// TIA Portal project "AGV75790" (V15)

(* hardware
DEVICE "ET 200S station_1"  ET 200S station
   slot 0: "Rack_0"  Rail
   slot 2: "PLC_AGV75790"  IM 151-8 PN/DP CPU  6ES7 151-8AB01-0AB0  V3.2
      slot 1: "PROFINET interface_1"  PN-IO
         slot 1: "Port_1"  Port
         slot 2: "Port_2"  Port
         slot 3: "Port_3"  Port
   slot 4: "PM-E 24VDC_1"  PM-E 24VDC  6ES7 138-4CA01-0AA0
   slot 5: "8DI x 24VDC_1"  8DI x 24VDC  6ES7 131-4BF00-0AA0
   slot 6: "2AO x U ST_1"  2AO x U ST  6ES7 135-4FB01-0AB0
   slot 7: "8DO x 24VDC / 0.5A_1"  8DO x 24VDC / 0.5A  6ES7 132-4BF00-0AA0
DEVICE "GSD device_1"  GSD.Device.PN
   slot 0: "Rack"  Rack  V1.0
   slot 0: "PGV_AGV75790"  PGVxxx-F200 Position Encoder Color DAP  PGVxxx-F200x-B17-V1D  V1.1.3
      slot 0: "PGVxxx-F200 Position Encoder Color DAP"  PGVxxx-F200 Position Encoder Color DAP
      slot 1: "Interface"  Interface
         slot 1: "Port 1"  Port 1
         slot 2: "Port 2"  Port 2
      slot 1: "Configuration"  Configuration
         slot 0: "Configuration"  Configuration
   slot 3: "status, y-postion, angle, x-position, z-distance"  status, y-postion, angle, x-position, z-distance
      slot 0: "status, y-postion, angle, x-position, z-distance"  status, y-postion, angle, x-position, z-distance
   slot 6: "Status Warning and Error"  Status Warning and Error
      slot 0: "Status Warning and Error"  Status Warning and Error
   slot 7: "input data"  input data
      slot 0: "input data"  input data
DEVICE "GSD device_2"  GSD.Device.PN
   slot 0: "Rack"  Rack  V1.0
   slot 0: "IOLINK_AGV75790"  BNI PNT-508-105-Z015  BNI005H  V3.2
      slot 0: "BNI PNT-508-105-Z015"  BNI PNT-508-105-Z015
      slot 1: "PN-IO"  PN-IO
         slot 1: "port 1 - M12"  port 1 - M12
         slot 2: "port 2 - M12"  port 2 - M12
      slot 1: "IOLINK_AGV72159_1"  BNI PNT-508-105-Z015
         slot 0: "BNI PNT-508-105-Z015"  BNI PNT-508-105-Z015
   slot 2: "MotorDePasso.08Bytes"  IOL_I/O_08/08 byte
      slot 0: "IOL_I/O_08/08 byte"  IOL_I/O_08/08 byte
   slot 3: "Rfid_Bis103"  IOL_I/O_32/32 byte
      slot 0: "IOL_I/O_32/32 byte"  IOL_I/O_32/32 byte
   slot 4: "Standard I/O_3"  Standard I/O
      slot 0: "Standard I/O"  Standard I/O
   slot 5: "Standard I/O_4"  Standard I/O
      slot 0: "Standard I/O"  Standard I/O
   slot 6: "Standard I/O_5"  Standard I/O
      slot 0: "Standard I/O"  Standard I/O
   slot 7: "Standard I/O_6"  Standard I/O
      slot 0: "Standard I/O"  Standard I/O
   slot 8: "Standard I/O_7"  Standard I/O
      slot 0: "Standard I/O"  Standard I/O
   slot 9: "Standard I/O_8"  Standard I/O
      slot 0: "Standard I/O"  Standard I/O
   slot 10: "Station diagnostic"  Station diagnostic
      slot 0: "Station diagnostic"  Station diagnostic
   slot 11: "Sensor supply short circuit"  Sensor supply short circuit
      slot 0: "Sensor supply short circuit"  Sensor supply short circuit
   slot 12: "Periphery error"  Periphery error
      slot 0: "Periphery error"  Periphery error
   slot 13: "Display Leds"  Display Leds
      slot 0: "Display Leds"  Display Leds
DEVICE "SCALANCE X005_1"  SCALANCE X-Station
   slot 0: "SCALANCE X rack"  Rail
   slot 0: "Switch_Rede"  6GK5 008-0GA00-1AB2  V1.0
DEVICE "HMI_AGV75790"  KTP600 Basic color PN
   slot 0: "HMI_AGV75790"  KTP600 Basic color PN  6AV6 647-0AD11-3AX0  12.0.0.0
   slot 1: "HMI_AGV72159"  KTP600 Basic color PN  6AV6 647-0AD11-3AX0  12.0.0.0
   slot 5: "HMI_AGV75790.IE_CP_1"  PROFINET Interface  12.0.0.0
      slot 1: "PROFINET Interface_1"  PROFINET Interface
         slot 1: "Port_1"  Port
*)

// ===== PLC "PLC_AGV75790"  IM 151-8 PN/DP CPU =====

VAR_GLOBAL   // PLC tag table "IO Link"
   "IOLink_StatusAGV" AT %IW80 : Word;   // Status do IOlink 0 - fora da rede, 1 - Na rede
END_VAR

VAR_GLOBAL   // PLC tag table "Entradas"
   "DI_BotaoStart" AT %I0.0 : Bool;   // Botão Wireless de Start do AGV
   "DI_Emergencia" AT %I0.1 : Bool;   // Botão de Emergencia
   "DI_Resevado" AT %I0.2 : Bool;   // Reservado/Sem utilidade no momento
   "DI_Resevado_1" AT %I0.3 : Bool;   // Reservado/Sem utilidade no momento
   "DI_ScannerWarning" AT %I0.4 : Bool;   // Sinal de atenção do Scanner de area
   "DI_ScannerSafety" AT %I0.5 : Bool;   // Sinal de Segurança do Scanner de area
   "DI_Resevado_2" AT %I0.6 : Bool;   // Reservado/Sem utilidade no momento
   "DI_Resevado_3" AT %I0.7 : Bool;   // Reservado/Sem utilidade no momento
END_VAR

VAR_GLOBAL   // PLC tag table "Saidas"
   "AO_MotorTracao" AT %QW752 : Int;   // Sinal de regulagem da velocidade do motor de tração
   "AO_Reservado" AT %QW754 : Int;   // Reservado/Sem utilidade no momento
   "DO_Reservado" AT %Q0.0 : Bool;   // Reservado/Sem utilidade no momento
   "DO_Reservado_1" AT %Q0.1 : Bool;   // Reservado/Sem utilidade no momento
   "DO_Motor.Frente" AT %Q0.2 : Bool;   // Sinal que controla o sentido de giro para frente do motor de tração
   "DO_Motor.Tras" AT %Q0.3 : Bool;   // Sinal que controla o sentido de giro para trás do motor de tração
   "DO_Scanner.Zone1" AT %Q0.4 : Bool;   // Sinal reservado para que seja possivel realizar o aumento e diminuição da area do Scanner de segurança
   "DO_Giroflex" AT %Q0.5 : Bool;   // Sinal luminoso do giroflex - Indica que o AGV está rodando
   "DO_Scanner.Zone2" AT %Q0.6 : Bool;   // Sinal reservado para que seja possivel realizar o aumento e diminuição da area do Scanner de segurança
   "DO_LuzReset" AT %Q0.7 : Bool;   // Sinal luminoso do de emergencia - Indica que o AGV está com o emergencia acionado
END_VAR

VAR_GLOBAL   // PLC tag table "ClockMemory"
   "ClockByte" AT %MB100 : Byte;   // Byte de Clock
   "Clock_10Hz" AT %M100.0 : Bool;   // 100 Milisegundos
   "Clock_5Hz" AT %M100.1 : Bool;   // 200 Milisegundos
   "Clock_2.5Hz" AT %M100.2 : Bool;   // 400 Milisegundos
   "Clock_2Hz" AT %M100.3 : Bool;   // 500 Milisegundos
   "Clock_1.25Hz" AT %M100.4 : Bool;   // 800 Milisegundos
   "Clock_1Hz" AT %M100.5 : Bool;   // 1 Segundos
   "Clock_0.625Hz" AT %M100.6 : Bool;   // 1,6 segundos
   "Clock_0.5Hz" AT %M100.7 : Bool;   // 2 Segundos
END_VAR

VAR_GLOBAL   // PLC tag table "Pgv_Tags"
   "ERR" AT %I1.0 : Bool;   // Error Message, See Error Codes
   "NP" AT %I1.1 : Bool;   // No Absolute Position
   "WRN" AT %I1.2 : Bool;   // Warning Present, See Warning Module
   "CC" AT %I1.3 : Bool;   // Control Code Detected
   "Reservado" AT %I1.4 : Bool;   // Reserved
   "FR" AT %I1.5 : Bool;   // Follow Right-hand lane
   "FL" AT %I1.6 : Bool;   // Follow Left-hand lane
   "NL" AT %I1.7 : Bool;   // No lane detected
   "RP" AT %I2.0 : Bool;   // Relative Position
   "LC" AT %I2.1 : Bool;   // Bit field LSB, Number of detected lanes
   "LC_1" AT %I2.2 : Bool;   // Bit field MSB, Number of detected lanes
   "TA" AT %I2.3 : Bool;   // Data Matrix tag present
   "Reservado_1" AT %I2.4 : Bool;   // Reserved
   "Reservado_2" AT %I2.5 : Bool;   // Reserved
   "Reservado_3" AT %I2.6 : Bool;   // Reserved
   "Reservado_4" AT %I2.7 : Bool;   // Reserved
   "PositionY" AT %ID3 : DWord;   // Posição no eixo Y
   "Angle" AT %IW8 : Word;   // Angulo
   "PositionX" AT %ID10 : DWord;   // Posição no eixo X
   "PositionZ" AT %IW14 : Word;   // Posição no eixo Z
   "Output_Data" AT %QB1 : Byte;   // Dados de Saida
   "Status" AT %ID15 : DWord;   // Status PGV
   "Erro" AT %IW20 : Word;   // Erros PGV
END_VAR

TYPE "DT_FML_STATUS"
VERSION : 0.1
   STRUCT
      Err : Bool;
      Cat : Int;
      ID : DInt;
   END_STRUCT;
END_TYPE

TYPE "DT_FML_PRM_FILE"
VERSION : 0.1
// DT_FML_PRM_FILE_TRANSFER
   STRUCT
      Control : Int;
      BitSequenceNr : Int;
      Data : Array[1..6] of Byte;
   END_STRUCT;
END_TYPE

TYPE "DT_FML_REF"
// DT_FML_PRM_REF
   STRUCT
      InData : Struct
         FHPP : Array[1..8] of Byte;
         FPC : Array[1..8] of Byte;
         FHPPplus : Array[1..10] of DInt;
      END_STRUCT;
      OutData : Struct
         FHPP : Array[1..8] of Byte;
         FPC : Array[1..8] of Byte;
         FHPPplus : Array[1..10] of DInt;
      END_STRUCT;
      Modbus : Bool;
      DeviceType : String[16];
      DeviceTypeNo : Byte;
      MemberID : Int;   // Current Axis-ID
      MemberIDmax : Int;   // Maximum Axis-ID
      Done : Bool;   // Execution Done
      Err : Bool;   // Fault occured
      PNU : Word;   // Number of the Parameter
      ActPNU : Word;   // Actual Number of the Parameter
      ReqID : Int;   // Read upper Limit of the Parameter
      RespID : Int;   // Read lower limit of the Parameter
      FPCC_Modus : Byte;   // modus of parameter channel control
      FPCS_Modus : Byte;   // modus of parameter channel status
      FPCC_Packet : "DT_FML_PRM_FILE";
      FPCS_Packet : "DT_FML_PRM_FILE";
      Subindex : Byte;   // Subindex of the Parameter to Exchange
      ActSubindex : Byte;   // Actual Subindex of the Parameter
      DatatypeWR : Byte;   // Length of the Parameter to Exchange in Byte
      DatatypeRD : Byte;   // Actual Length of the Parameter in Byte
      ParamValueWR : DInt;   // Value of the Parameter to Exchange
      ParamValueRD : DInt;   // Read Value of Parameter
   END_STRUCT;
END_TYPE

TYPE "EscritaTakt"
   STRUCT
      Emergencia : Bool;   // Botao de Emergecencia
      Warning : Bool;   // Area de Warning do Scanner
      Safety : Bool;   // Area de Safety do Scanner
      ConectarTakt : Bool;   // 0 - Desconectado / 1 - Conectado
      Rodando : Bool;
      Falha : Bool;
      AutomaticoManual : Byte;   // 1 - Manual / 2 - Automatico
      VelocidadeAtual : Int;   // Velocidade Atual
      Posto : Byte;   // Posto em que o AGV está
      Comando : Byte;   // Ultimo comando
      Velocidade : Byte;   // Velocidade Setada
      Processo : Byte;   // 1 - Ecu / 2 - SKD
      "Erros.Agv" : Byte;   // 0 á 256, cada numero um erro. 1 - Tudo Ok
      "Erros.Pgv" : Byte;   // 0 á 256, cada numero um erro. 1 - Tudo Ok
      "Erros.Rfid" : Byte;   // 0 á 256, cada numero um erro. 1 - Tudo Ok
      "Erros.MotorPasso" : Byte;   // 0 á 256, cada numero um erro. 1 - Tudo Ok
      "Erros.IOLink" : Byte;   // 0 á 256, cada numero um erro. 1 - Tudo Ok
      "Erros.Comunicacao" : Byte;   // 0 á 256, cada numero um erro. 1 - Tudo Ok
      Reservado : Byte;   // Reservado
      Reservado_1 : Byte;   // Reservado
      Reservado_2 : Byte;   // Reservado
      Reservado_3 : Byte;   // Reservado
      Reservado_4 : Byte;   // Reservado
      Reservado_5 : Byte;   // Reservado
      Reservado_6 : Byte;   // Reservado
      Reservado_7 : Byte;   // Reservado
      Reservado_8 : Byte;   // Reservado
   END_STRUCT;
END_TYPE

TYPE "LeituraTakt"
   STRUCT
      EmergenciaECU : Bool;   // Emergencia
      EmergenciaSKD : Bool;   // Emergencia
      StartAgvECU : Bool;   // Start by takt
      StopAgvECU : Bool;   // Stop by takt
      StartAgvSKD : Bool;   // Start by takt
      StopAgvSKD : Bool;   // Stop by takt
      WatchDog : Bool;   // WatchDog
      TOD : Time_Of_Day;   // Time of day
   END_STRUCT;
END_TYPE

// folder: 01_Controle/02_DB

DATA_BLOCK "DB1_DatabaseAgv"   // DB1
TITLE = DB1_DatabaseAgv
{ S7_Optimized_Access := 'FALSE' }
AUTHOR : ssbjvq
VERSION : 0.1
// Está DB é responsavel por centralizar toda a informação do AGV
   VAR
      Entradas : Struct   // Sinais do cartão de entrada digital
         BotaoStart : Bool;   // Botão Wireless de Start do AGV
         BotaoEmergencia : Bool;   // Botão de Emergencia
         ScannerWarning : Bool;   // Sinal de atenção do Scanner de area
         ScannerSafety : Bool;   // Sinal de Segurança do Scanner de area
         Reservada_4 : Bool;   // Reservado/Sem utilidade no momento
         Reservada_5 : Bool;   // Reservado/Sem utilidade no momento
         Reservada_6 : Bool;   // Reservado/Sem utilidade no momento
      END_STRUCT;
      Saidas : Struct   // Sinais dos cartões de saida
         MotorFrente : Bool;   // Sinal que controla o sentido de giro para frente do motor de tração
         MotorTras : Bool;   // Sinal que controla o sentido de giro para trás do motor de tração
         Zona1_Scanner : Bool;   // Sinal reservado para que seja possivel realizar o aumento e diminuição da area do Scanner de segurança
         Zona2_Scanner : Bool;   // Sinal luminoso do giroflex - Indica que o AGV está rodando
         Giroflex : Bool;   // Sinal reservado para que seja possivel realizar o aumento e diminuição da area do Scanner de segurança
         LuzReset : Bool;   // Sinal luminoso do de emergencia - Indica que o AGV está com o emergencia acionado
         Reservada : Bool;   // Reservado/Sem utilidade no momento
         VelocidadeMotorTracao : Int;   // Sinal de regulagem da velocidade do motor de tração
         Analog_1 : Int;   // Reservado/Sem utilidade no momento
      END_STRUCT;
      PGV : Struct   // Sinais do PGV
         Module2 : Struct
            Status : Struct
               ERR : Bool;   // Error Message, See Error Codes
               NP : Bool;   // No Absolute Position
               WRN : Bool;   // Warning Present, See Warning Module
               CC : Bool;   // Control Code Detected
               Reservado : Bool;   // Reserved
               FR : Bool;   // Follow Right-hand lane
               FL : Bool;   // Follow Left-hand lane
               NL : Bool;   // No lane detected
               RP : Bool;   // Relative Position
               LC : Bool;   // Bit field LSB, Number of detected lanes
               LC_1 : Bool;   // Bit field MSB, Number of detected lanes
               TA : Bool;   // Data Matrix tag present
               Reservado_1 : Bool;   // Reserved
               Reservado_2 : Bool;   // Reserved
               Reservado_3 : Bool;   // Reserved
               Reservado_4 : Bool;   // Reserved
            END_STRUCT;
            PositionY : DWord;
            Angle : Word;
            PositionX : DWord;
            PositionZ : Word;
         END_STRUCT;
         Module5 : Struct
            Status : Word;
            BitmaskWarning : Word;
            ErroNumber : Word;
         END_STRUCT;
         Mensagens : String;
         NaRota : Bool;
         Rota : Byte := 16#0A;
      END_STRUCT;
      RFID : Struct   // Sinais do RFID
         Inputs : Struct
            Init : Bool;   // Deve ser pulsado para iniciar a leitura
            Start : Bool;   // Deve ser dado o start para o RIFD funcionar
            Reset : Bool;   // Reseta se existe problema
            HeadOff : Bool;
            Dynamic : Bool;
            HW_IO : Int := 80;   // Endereço do dispositivo na rede
            Command : Int := 1;   // Comando 1 - Leitura / 2 - Escrita
            DB_Send : Int := 421;   // Numero da DB de envio de dados
            Offset_DBSend : Int := 0;   // Deslocamento de bits da DB de envio
            DB_Receive : Int := 420;   // Numero da DB de recebimento de dados
            Offset_DBReceive : Int := 0;   // Deslocamento de bits da DB de recebimento
            StartAddress : Int := 0;   // Primeiro endereço a ser lido
            NumberOfByte : Int := 32;   // Numero de bytes a ser lidos até 32 bits
            Watchdog : S5Time := S5T#100ms;
         END_STRUCT;
         Posto : Int;   // Valor do posto
         Comando : Int;   // Valor do comando
         Velocidade : Int := 22;   // Valor da velocidade
         Processo : Int;   // Valor da linha
         Error : Bool;   // Sinal de erro
         TagPresente : Bool;   // Sinal de Tag presente
         CodigoErro : Int;   // Codigo do erro
         Ready : Bool;   // Sinal de Pronto para uso
         Fault : Bool;   // Sinal de falha
         Mensagens : String;   // Mensagens de falha
      END_STRUCT;
      MotorDePasso : Struct   // Sinais do Motor de Passo
         GetIO : Struct   // Bloco de comunicação
            Inputs : Struct
               IAddress_FHPP : Word := 16#46;   // Endereço do dispositivo em HEX
               Offset : Int := 0;   // Deslocamento de bits
               DeviceType : String[16] := 'CMMO_ST';   // Tipo do dispositivo
            END_STRUCT;
            Outputs : Struct
               Error : Bool;   // Sinal de falha na comunicação
               Status : "DT_FML_STATUS";   // Status de leitura
            END_STRUCT;
         END_STRUCT;
         SetIO : Struct   // Bloco de comunicação
            Inputs : Struct
               ID : Word := 16#46;   // Endereço do dispositivo em HEX
               Offset : Int;   // Deslocamento de bits
            END_STRUCT;
            Outputs : Struct
               Error : Bool;   // Sinal de falha na comunicação
               Status : "DT_FML_STATUS";   // Status de leitura
            END_STRUCT;
         END_STRUCT;
         Inputs : Struct   // Sinais de entrada
            EnableDrive : Bool;   // Habilitar drive
            Stop : Bool;   // Parar motor
            Halt : Bool;
            Brake : Bool;   // Freio do motor
            ResetFault : Bool;   // Resetar falha do motor
            HMIAccessLocked : Bool;   // Travar acesso via IHM
            OPM : Int;   // Modo de operação
            StartTask : Bool;   // Iniciar tarefa
            StartHoming : Bool;   // Iniciar homing
            JogPos : Bool;   // Virar a esquerda
            JogNeg : Bool;   // Virar a direita
            TeachActValue : Bool;
            ClearRemPos : Bool;
            Relative : Bool;
            DeactivateStrokeLimit : Bool;   // Desativar limite de giro
            ExecuteFunction : Bool;   // Executar função gravada
            RecordNo : Int;   // Numero da função
            SetFunctionNumber : Int;   // Setar numero da função
            SetFunctionGroup : Int;   // Setar numero do grupo de funções
            SetValueVelocity : DInt;   // Setar valor de velocidade do motor
            SetValuePosition : DInt;   // Setar valor de posição
            SetValueForceRamp : DInt;   // Setar valor de rampa de força
            SetValueForce : DInt;   // Setar valor de força
            SetValueRotRamp : DInt;   // Setar valor de rampa de rotação
            SetValueRotSpeed : DInt;   // Setar valor de rotação
         END_STRUCT;
         OutPuts : Struct   // Sinais de saidas
            DriveEnabled : Bool;   // Drive habilitado
            Ready : Bool;   // Pronto para rodar
            Warning : Bool;   // Em modo atenção
            Fault : Bool;   // Em falha
            SupplyVoltPresent : Bool;   // Tensão presente
            ControlFCT_HMI : Bool;   // Controle via IHM
            StateOPM : Int;   // Status do modo de operação
            HaltNotActive : Bool;   // Halt não ativado
            AckStart : Bool;   // Movimento iniciado
            MC : Bool;   // Movimento Completo
            AckTeach : Bool;
            DriveMoving : Bool;   // Motor em movimento
            DragError : Bool;   // Error de movimentação
            StandStillControl : Bool;
            HomingValid : Bool;   // Homing valido
            ActualRecordNo : Int;   // Numero de gravação atual
            RC1 : Bool;
            RCC : Bool;
            VelocityLimitReached : Bool;   // Velocidade limite atingida
            StrokeLimitReached : Bool;   // Giro limite atingido
            FunctionIsActive : Bool;   // Modo função ativado
            ActualFunctionNumber : Int;   // Numero atual da função
            ActualFunctionGroup : Int;   // Numero atual do grupo de função
            ActualPosition : DInt;   // Posição atual
            ActualVelocity : Int;   // Velocidade atual
            ActualForce : Int;   // Força atual
            ActualRotRamp : Int;   // Rampa de rotação atual
            ActualRotSpeed : DInt;   // Velocidade de rotação atual
         END_STRUCT;
         Mensagens : String;   // Mensagens de motor de passo
      END_STRUCT;
      IOLink : Struct   // Sinais do IOLink
         Mensagens : String;   // Mensagens de falha do IO Link
      END_STRUCT;
      Takt : Struct   // Sinais do Takt
         Mensagens : String;
      END_STRUCT;
      Mensagens : String;   // Mensagens gerais do AGV
   END_VAR
BEGIN
END_DATA_BLOCK

DATA_BLOCK "DB3_Memorias"   // DB3
{ S7_Optimized_Access := 'FALSE' }
VERSION : 0.1
   VAR
      StartStop : Bool;   // Memoria de Start ou Stop
      Rfid : Struct   // Memorias do RFId
         PararAgv : Bool;   // Memoria de parada do AGV
         Comando : Int;   // Memoria de comando
         Velocidade : Int;   // Memoria de velocidade
         Linha : Int;   // Memoria de linha
         Posto : Int;   // Memoria de posto
         LeituraEscrita : Int;   // Memoria de leitura 1 ou escrita 2
      END_STRUCT;
      Pgv : Struct   // Memorias do Pgv
         NaRota : Bool;   // AGV na rota
         Angulo : Int;   // Angulo
         Direita : Bool;   // Direita
         Esquerda : Bool;   // Esquerda
      END_STRUCT;
      Frente : Bool;
      Tras : Bool;
      Esquerda : Bool;
      Direita : Bool;
      Posicao : DInt;   // Posição motor de passo
      Velocidade : Int;   // Velocidade
      EmCurva : Bool;   // Memoria Em curva
      EmCurvaIntermediario : Bool;   // Memoria Em curva intermediario
      LimiteGiroDireita : Bool;   // Bloco de comunicação
      LimiteGiroEsquerda : Bool;   // Memoria de limite de giro
   END_VAR
BEGIN
END_DATA_BLOCK

DATA_BLOCK "DB100_ManualAutomatico_DB"   // DB100
{ S7_Optimized_Access := 'FALSE' }
VERSION : 0.1
// stored: InstanceOfName FB100_ManualAutomatico
"FB100_ManualAutomatico"
BEGIN
END_DATA_BLOCK

DATA_BLOCK "DB102_AgvStartStop"   // DB102
{ S7_Optimized_Access := 'FALSE' }
VERSION : 0.1
// stored: InstanceOfName FB102_AgvStartStop
"FB102_AgvStartStop"
BEGIN
END_DATA_BLOCK

DATA_BLOCK "DB105_Sinalizacao"   // DB105
{ S7_Optimized_Access := 'FALSE' }
VERSION : 0.1
// stored: InstanceOfName FB105_Sinalizacao
"FB105_Sinalizacao"
BEGIN
END_DATA_BLOCK

// folder: 02_MotorPasso/02_DB

DATA_BLOCK "DB200_ControleMotorDePasso"   // DB200
{ S7_Optimized_Access := 'FALSE' }
VERSION : 0.1
// stored: InstanceOfName FB200_ControleMotorDePasso
"FB200_ControleMotorDePasso"
BEGIN
END_DATA_BLOCK

// folder: 03_Pgv/02_DB

DATA_BLOCK "DB301_PgvDados"   // DB4
{ S7_Optimized_Access := 'FALSE' }
VERSION : 0.1
// stored: InstanceOfName FB301_PgvDados
"FB301_PgvDados"
BEGIN
END_DATA_BLOCK

DATA_BLOCK "DB300_LogicaPgv"   // DB300
{ S7_Optimized_Access := 'FALSE' }
VERSION : 0.1
// stored: InstanceOfName FB300_LogicaPgv
"FB300_LogicaPgv"
BEGIN
END_DATA_BLOCK

// folder: 04_Rfid/02_DB

DATA_BLOCK "DB400_LogicaRfid"   // DB400
{ S7_Optimized_Access := 'FALSE' }
VERSION : 0.1
// stored: InstanceOfName FB400_LogicaRfid
"FB400_LogicaRfid"
BEGIN
END_DATA_BLOCK

DATA_BLOCK "DB420_LeituraRfid"   // DB420
{ S7_Optimized_Access := 'FALSE' }
VERSION : 0.1
   VAR
      RfidLeitura : Array[0..31] of Int;
   END_VAR
BEGIN
   RfidLeitura[3] := 22;   // Velocidade
   RfidLeitura[1] := 2;   // Posto de trabalho
   // RfidLeitura[2] : Comando
   // RfidLeitura[4] : Linha/Processo
   // RfidLeitura[0] : Não utilizado
   // RfidLeitura[5] : Não utilizado
   // RfidLeitura[6] : Não utilizado
   // RfidLeitura[7] : Não utilizado
   // RfidLeitura[8] : Não utilizado
   // RfidLeitura[9] : Não utilizado
   // RfidLeitura[10] : Não utilizado
   // RfidLeitura[11] : Não utilizado
   // RfidLeitura[12] : Não utilizado
   // RfidLeitura[13] : Não utilizado
   // RfidLeitura[14] : Não utilizado
   // RfidLeitura[15] : Não utilizado
   // RfidLeitura[16] : Não utilizado
   // RfidLeitura[17] : Não utilizado
   // RfidLeitura[18] : Não utilizado
   // RfidLeitura[19] : Não utilizado
   // RfidLeitura[20] : Não utilizado
   // RfidLeitura[21] : Não utilizado
   // RfidLeitura[22] : Não utilizado
   // RfidLeitura[23] : Não utilizado
   // RfidLeitura[24] : Não utilizado
   // RfidLeitura[25] : Não utilizado
   // RfidLeitura[26] : Não utilizado
   // RfidLeitura[27] : Não utilizado
   // RfidLeitura[28] : Não utilizado
   // RfidLeitura[29] : Não utilizado
   // RfidLeitura[30] : Não utilizado
   // RfidLeitura[31] : Não utilizado
END_DATA_BLOCK

DATA_BLOCK "DB421_EscritaRfid"   // DB421
{ S7_Optimized_Access := 'FALSE' }
VERSION : 0.1
   VAR
      RfidEscrita : Array[0..31] of Int;
   END_VAR
BEGIN
   // RfidEscrita[0] : Não utilizado
   // RfidEscrita[1] : Posto de trabalho
   // RfidEscrita[2] : Comando
   // RfidEscrita[3] : Velocidade
   // RfidEscrita[4] : Linha/Processo
   // RfidEscrita[5] : Não utilizado
   // RfidEscrita[6] : Não utilizado
   // RfidEscrita[7] : Não utilizado
   // RfidEscrita[8] : Não utilizado
   // RfidEscrita[9] : Não utilizado
   // RfidEscrita[10] : Não utilizado
   // RfidEscrita[11] : Não utilizado
   // RfidEscrita[12] : Não utilizado
   // RfidEscrita[13] : Não utilizado
   // RfidEscrita[14] : Não utilizado
   // RfidEscrita[15] : Não utilizado
   // RfidEscrita[16] : Não utilizado
   // RfidEscrita[17] : Não utilizado
   // RfidEscrita[18] : Não utilizado
   // RfidEscrita[19] : Não utilizado
   // RfidEscrita[20] : Não utilizado
   // RfidEscrita[21] : Não utilizado
   // RfidEscrita[22] : Não utilizado
   // RfidEscrita[23] : Não utilizado
   // RfidEscrita[24] : Não utilizado
   // RfidEscrita[25] : Não utilizado
   // RfidEscrita[26] : Não utilizado
   // RfidEscrita[27] : Não utilizado
   // RfidEscrita[28] : Não utilizado
   // RfidEscrita[29] : Não utilizado
   // RfidEscrita[30] : Não utilizado
   // RfidEscrita[31] : Não utilizado
END_DATA_BLOCK

// folder: 05_Ihm/02_DB

DATA_BLOCK "DB500_SinaisIhm"   // DB500
{ S7_Optimized_Access := 'FALSE' }
VERSION : 0.1
   VAR
      ManualAutomatico : Int := 1;   // 1 Modo manual/ 2 - modo automatico
      Start : Bool;   // Botão de Start IHM
      Processo : Int := 1;   // Botão de processo IHM
      VelocidadeManual : Int := 18;   // Velocidade em manual
      VelocidadeWarning : Int := 10;   // Velocidade em Warning
      ResetFault : Bool;   // Botao de Resetar falha do motor
      ManFrente : Bool;   // Botao manual frente
      ManTras : Bool;   // Botao manual tras
      ManDireita : Bool;   // Botao manual direita
      ManEsquerda : Bool;   // Botao manual esquerda
      ConexaoTakt : Bool := TRUE;   // Conectar com o takt
      PostoRfid : Int;   // Input de gravação de tag
      ComandoRfid : Int;   // Input de gravação de tag
      VelocidadeRfid : Int;   // Input de gravação de tag
      ProcessoRfid : Int;   // Input de gravação de tag
      LeituraEscritaRfid : Bool;   // Modo de operação do RFID
      VelocidadeAutomatico : Int := 15;   // Valor de velocidade em automatico
      VelocidadeAtual : Int;   // Valor de velocidade atual
      ConectarTakt : Int := 1;   // 1 - Conecta com o Takt / 0 - Desconectado
      ResetFalha_Rfid : Bool := False;   // Resetar falha RFID
   END_VAR
BEGIN
END_DATA_BLOCK

// folder: 06_Errors/02_DB

DATA_BLOCK "DB600_AgvSinais"   // DB600
{ S7_Optimized_Access := 'FALSE' }
VERSION : 0.1
   VAR
      Inputs : Struct   // Cartão de entrada
         "8DI_24V" : Struct   // Cartão de entrada
            "I0.0" : Bool;   // Botão Wireless de Start do AGV
            "I0.1" : Bool;   // Botão de Emergencia
            "I0.2" : Bool;   // Reservado/Sem utilidade no momento
            "I0.3" : Bool;   // Reservado/Sem utilidade no momento
            "I0.4" : Bool;   // Sinal de atenção do Scanner de area
            "I0.5" : Bool;   // Sinal de Segurança do Scanner de area
            "I0.6" : Bool;   // Reservado/Sem utilidade no momento
            "I0.7" : Bool;   // Reservado/Sem utilidade no momento
         END_STRUCT;
      END_STRUCT;
      Outputs : Struct   // Cartões de saida
         "8DO_24V" : Struct   // Cartão Digital
            "Q0.0" : Bool;   // Reservado/Sem utilidade no momento
            "Q0.1" : Bool;   // Reservado/Sem utilidade no momento
            "Q0.2" : Bool;   // Sinal que controla o sentido de giro para frente do motor de tração
            "Q0.3" : Bool;   // Sinal que controla o sentido de giro para trás do motor de tração
            "Q0.4" : Bool;   // Sinal reservado para que seja possivel realizar o aumento e diminuição da area do Scanner de segurança
            "Q0.5" : Bool;   // Sinal luminoso do giroflex - Indica que o AGV está rodando
            "Q0.6" : Bool;   // Sinal reservado para que seja possivel realizar o aumento e diminuição da area do Scanner de segurança
            "Q0.7" : Bool;   // Sinal luminoso do de emergencia - Indica que o AGV está com o emergencia acionado
         END_STRUCT;
         "2AO x U ST" : Struct   // Cartão Analogico
            QW750 : Word;   // Sinal de regulagem da velocidade do motor de tração
            QW752 : Word;   // Reservado/Sem utilidade no momento
         END_STRUCT;
      END_STRUCT;
      RFID : Struct   // Sinais RFID
         Posto : Int;   // Valor do posto
         Comando : Int;   // Valor do comando
         Velocidade : Int;   // Valor da velocidade
         Linha : Int;   // Valor da linha
         Tag_Presente : Bool;   // Sinal de erro
         Error : Bool;   // Sinal de Tag presente
         Code_Error : Int;   // Codigo do erro
         Ready : Bool;   // Sinal de Pronto para uso
         Mensagem : String;   // Sinal de falha
      END_STRUCT;
      Stepping_Motor : Struct   // Sinais Motor de Passo
         Inputs : Struct   // Entrada
            Enabla_Drive : Bool;   // Habilitar Dirve
            Stop : Bool;   // Parado
            "Start Task" : Bool;   // Inicia Tarefa
            Opm : Int;   // Modo de operação
            Brake : Bool;   // Freio
         END_STRUCT;
         Outputs : Struct   // Saidas
            DriveEnabled : Bool;   // Drive habilitado
            Ready : Bool;   // Pronto para rodar
            Warning : Bool;   // Em modo atenção
            Fault : Bool;   // Em falha
            SupplyVoltPresent : Bool;   // Tensão presente
            DragError : Bool;   // Error de movimentação
            HomingValid : Bool;   // Homing valido
            StrokeLimitReached : Bool;   // Giro limite atingido
            ActualPosition : DInt;   // Posição atual
         END_STRUCT;
         Mensagem : String;   // Mensagens do motor de passo
      END_STRUCT;
      PGV : Struct   // Sinais PGV
         Mensagem : String;   // Mensagens do PGV
         ERR : Bool;   // Error Message, See Error Codes
         NP : Bool;   // No Absolute Position
         WRN : Bool;   // Warning Present, See Warning Module
         CA : Bool;   // Control Code Detected
         FR : Bool;   // Reserved
         FL : Bool;   // Follow Right-hand lane
         NL : Bool;   // Follow Left-hand lane
         RP : Bool;   // No lane detected
         TA : Bool;   // Relative Position
         PositionData_Y : Int;   // Bit field LSB, Number of detected lanes
         PositionData_X : Int;   // Bit field MSB, Number of detected lanes
         PositionData_Z : Int;   // Data Matrix tag present
         AngleData : Int;   // Angulo
         "DataMatrix.CCStatus" : Byte;
         "DataMatrix.CCNumber" : Word;
         "DataMatrix.TagNumber" : DWord;
         BitmaskWarning : Word;
         ErrorNumber : Word;
         "OUT_Warning.Monitoring" : Word;
         "OUT_Error.Monitoring" : Word;
      END_STRUCT;
      DateHora : Date_And_Time;   // Data e Hora
      Mensagens_Global : String;   // Mensagens de falha
      Alarms : Array[0..8] of Int;   // Alarmes na lista
   END_VAR
BEGIN
   // Alarms[0] : PGV
   // Alarms[1] : RFID
   // Alarms[2] : MOTOR DE PASSO
   // Alarms[3] : PLC
   // Alarms[4] : IO-LINK
   // Alarms[5] : SINAIS - 0 - Emergencia, 1 - Warning, 2- Safety, 3 - Fora da rota,
END_DATA_BLOCK

DATA_BLOCK "DB603_StatusGeralAgv"   // DB603
{ S7_Optimized_Access := 'FALSE' }
VERSION : 0.1
// stored: InstanceOfName FB603_StatusGeralAgv
"FB603_StatusGeralAgv"
BEGIN
END_DATA_BLOCK

// folder: 07_Takt/02_DB

DATA_BLOCK "DB700_EnviaDados"   // DB700
TITLE = DB700_EnviaDados
{ S7_Optimized_Access := 'FALSE' }
AUTHOR : ssbjvq
VERSION : 0.1
// DB700_EnviaDados
   VAR
      Dados : "EscritaTakt";
   END_VAR
BEGIN
END_DATA_BLOCK

DATA_BLOCK "DB701_RecebeDados"   // DB701
TITLE = DB701_RecebeDados
{ S7_Optimized_Access := 'FALSE' }
AUTHOR : ssbjvq
VERSION : 0.1
// DB701_RecebeDados
   VAR
      Dados : "LeituraTakt";
   END_VAR
BEGIN
END_DATA_BLOCK

DATA_BLOCK "DB703_ControleTakt"   // DB703
{ S7_Optimized_Access := 'FALSE' }
AUTHOR : ssbjvq
VERSION : 0.1
// stored: InstanceOfName FB703_ControleTakt
"FB703_ControleTakt"
BEGIN
END_DATA_BLOCK

DATA_BLOCK "DB704_DadosTakt"   // DB704
{ S7_Optimized_Access := 'FALSE' }
VERSION : 0.1
   VAR
      Dados_Takt : Struct
         Tempo_Takt : DInt;
         Tempo_StopTime : DInt;
         Objetivo : Int;
         Atual : Int;
         Andons : Array[0..8] of Bool;
      END_STRUCT;
   END_VAR
BEGIN
END_DATA_BLOCK

// folder: (top level)

ORGANIZATION_BLOCK "Main"   // OB1, LAD
TITLE = "Main Program Sweep (Cycle)"
{ S7_Optimized_Access := 'FALSE' }
VERSION : 0.1
// Bloco principal do CLP, ele é responsavel por rodar toda a logica do CLP e organizar o programa.
   VAR_TEMP
      OB1_EV_CLASS : Byte;   // Bits 0-3 = 1 (Coming event), Bits 4-7 = 1 (Event class 1)
      OB1_SCAN_1 : Byte;   // 1 (Cold restart scan 1 of OB 1), 3 (Scan 2-n of OB 1)
      OB1_PRIORITY : Byte;   // Priority of OB Execution
      OB1_OB_NUMBR : Byte;   // 1 (Organization block 1, OB1)
      OB1_RESERVED_1 : Byte;   // Reserved for system
      OB1_RESERVED_2 : Byte;   // Reserved for system
      OB1_PREV_CYCLE : Int;   // Cycle time of previous OB1 scan (milliseconds)
      OB1_MIN_CYCLE : Int;   // Minimum cycle time of OB1 (milliseconds)
      OB1_MAX_CYCLE : Int;   // Maximum cycle time of OB1 (milliseconds)
      OB1_DATE_TIME : Date_And_Time;   // Date and time OB1 started
   END_VAR
BEGIN

REGION Network 1: Modo Automatico ou Manual
   // Este bloco é responsavel por realizar o controle do AGV no modo automatico e no modo manual, sem ele o AGV não realiza nenhum movimento.
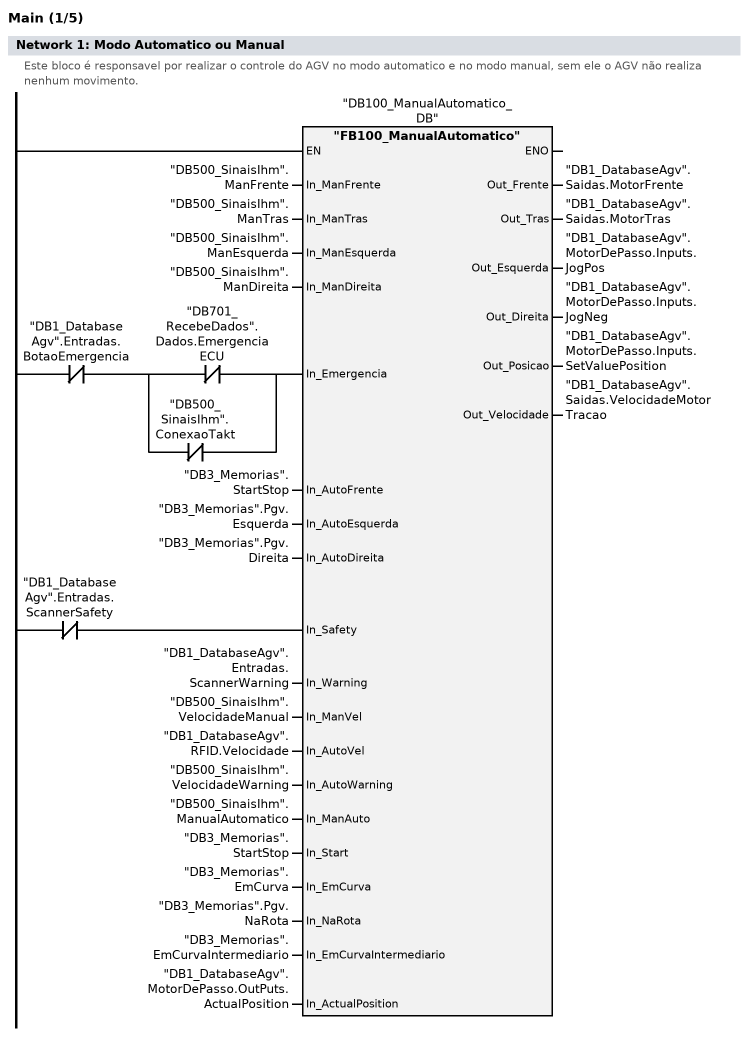
   RUNG wire#powerrail
      "DB100_ManualAutomatico_DB"(In_Emergencia := wire#w2, In_Safety := wire#w3, In_ManFrente := "DB500_SinaisIhm".ManFrente, In_ManTras := "DB500_SinaisIhm".ManTras, In_ManEsquerda := "DB500_SinaisIhm".ManEsquerda, In_ManDireita := "DB500_SinaisIhm".ManDireita, In_AutoFrente := "DB3_Memorias".StartStop, In_AutoEsquerda := "DB3_Memorias".Pgv.Esquerda, In_AutoDireita := "DB3_Memorias".Pgv.Direita, In_Warning := "DB1_DatabaseAgv".Entradas.ScannerWarning, In_ManVel := "DB500_SinaisIhm".VelocidadeManual, In_AutoVel := "DB1_DatabaseAgv".RFID.Velocidade, In_AutoWarning := "DB500_SinaisIhm".VelocidadeWarning, In_ManAuto := "DB500_SinaisIhm".ManualAutomatico, In_Start := "DB3_Memorias".StartStop, In_EmCurva := "DB3_Memorias".EmCurva, In_NaRota := "DB3_Memorias".Pgv.NaRota, In_EmCurvaIntermediario := "DB3_Memorias".EmCurvaIntermediario, In_ActualPosition := "DB1_DatabaseAgv".MotorDePasso.OutPuts.ActualPosition, Out_Frente => "DB1_DatabaseAgv".Saidas.MotorFrente, Out_Tras => "DB1_DatabaseAgv".Saidas.MotorTras, Out_Esquerda => "DB1_DatabaseAgv".MotorDePasso.Inputs.JogPos, Out_Direita => "DB1_DatabaseAgv".MotorDePasso.Inputs.JogNeg, Out_Posicao => "DB1_DatabaseAgv".MotorDePasso.Inputs.SetValuePosition, Out_Velocidade => "DB1_DatabaseAgv".Saidas.VelocidadeMotorTracao)
   END_RUNG
   RUNG wire#powerrail
      I_Contact( "DB1_DatabaseAgv".Entradas.BotaoEmergencia )
      wire#w1
      I_Contact( "DB701_RecebeDados".Dados.EmergenciaECU )
   END_RUNG wire#w2
   RUNG wire#w1
      I_Contact( "DB500_SinaisIhm".ConexaoTakt )
   END_RUNG wire#w2
   RUNG wire#powerrail
      I_Contact( "DB1_DatabaseAgv".Entradas.ScannerSafety )
   END_RUNG wire#w3
   // the same network as SCL:
   "DB100_ManualAutomatico_DB"(In_ManFrente := "DB500_SinaisIhm".ManFrente,   // "FB100_ManualAutomatico"
                           In_ManTras := "DB500_SinaisIhm".ManTras,
                           In_ManEsquerda := "DB500_SinaisIhm".ManEsquerda,
                           In_ManDireita := "DB500_SinaisIhm".ManDireita,
                           In_Emergencia := NOT "DB1_DatabaseAgv".Entradas.BotaoEmergencia AND (NOT "DB701_RecebeDados".Dados.EmergenciaECU OR NOT "DB500_SinaisIhm".ConexaoTakt),
                           In_AutoFrente := "DB3_Memorias".StartStop,
                           In_AutoEsquerda := "DB3_Memorias".Pgv.Esquerda,
                           In_AutoDireita := "DB3_Memorias".Pgv.Direita,
                           In_Safety := NOT "DB1_DatabaseAgv".Entradas.ScannerSafety,
                           In_Warning := "DB1_DatabaseAgv".Entradas.ScannerWarning,
                           In_ManVel := "DB500_SinaisIhm".VelocidadeManual,
                           In_AutoVel := "DB1_DatabaseAgv".RFID.Velocidade,
                           In_AutoWarning := "DB500_SinaisIhm".VelocidadeWarning,
                           In_ManAuto := "DB500_SinaisIhm".ManualAutomatico,
                           In_Start := "DB3_Memorias".StartStop,
                           In_EmCurva := "DB3_Memorias".EmCurva,
                           In_NaRota := "DB3_Memorias".Pgv.NaRota,
                           In_EmCurvaIntermediario := "DB3_Memorias".EmCurvaIntermediario,
                           In_ActualPosition := "DB1_DatabaseAgv".MotorDePasso.OutPuts.ActualPosition,
                           Out_Frente => "DB1_DatabaseAgv".Saidas.MotorFrente,
                           Out_Tras => "DB1_DatabaseAgv".Saidas.MotorTras,
                           Out_Esquerda => "DB1_DatabaseAgv".MotorDePasso.Inputs.JogPos,
                           Out_Direita => "DB1_DatabaseAgv".MotorDePasso.Inputs.JogNeg,
                           Out_Posicao => "DB1_DatabaseAgv".MotorDePasso.Inputs.SetValuePosition,
                           Out_Velocidade => "DB1_DatabaseAgv".Saidas.VelocidadeMotorTracao);
END_REGION

REGION Network 2: Logica do RFID
   // Este bloco controla do a logica de valores de parada, velocidade e posto. estes valores são lidos de um cartão RFID pela antena RFID no AGV.
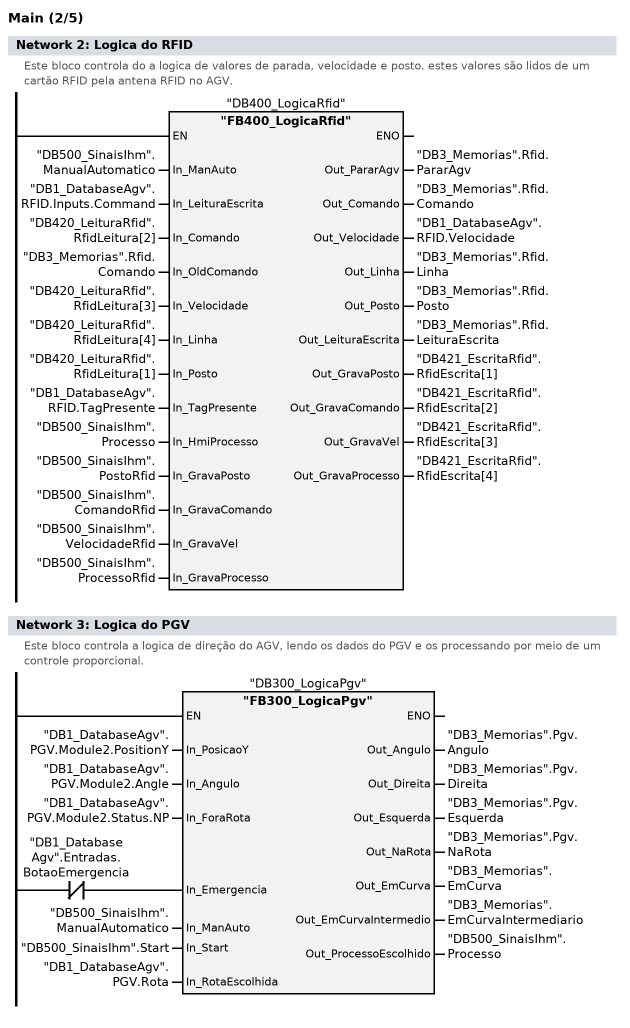
   RUNG wire#powerrail
      "DB400_LogicaRfid"(In_ManAuto := "DB500_SinaisIhm".ManualAutomatico, In_LeituraEscrita := "DB1_DatabaseAgv".RFID.Inputs.Command, In_Comando := "DB420_LeituraRfid".RfidLeitura[2], In_OldComando := "DB3_Memorias".Rfid.Comando, In_Velocidade := "DB420_LeituraRfid".RfidLeitura[3], In_Linha := "DB420_LeituraRfid".RfidLeitura[4], In_Posto := "DB420_LeituraRfid".RfidLeitura[1], In_TagPresente := "DB1_DatabaseAgv".RFID.TagPresente, In_HmiProcesso := "DB500_SinaisIhm".Processo, In_GravaPosto := "DB500_SinaisIhm".PostoRfid, In_GravaComando := "DB500_SinaisIhm".ComandoRfid, In_GravaVel := "DB500_SinaisIhm".VelocidadeRfid, In_GravaProcesso := "DB500_SinaisIhm".ProcessoRfid, Out_PararAgv => "DB3_Memorias".Rfid.PararAgv, Out_Comando => "DB3_Memorias".Rfid.Comando, Out_Velocidade => "DB1_DatabaseAgv".RFID.Velocidade, Out_Linha => "DB3_Memorias".Rfid.Linha, Out_Posto => "DB3_Memorias".Rfid.Posto, Out_LeituraEscrita => "DB3_Memorias".Rfid.LeituraEscrita, Out_GravaPosto => "DB421_EscritaRfid".RfidEscrita[1], Out_GravaComando => "DB421_EscritaRfid".RfidEscrita[2], Out_GravaVel => "DB421_EscritaRfid".RfidEscrita[3], Out_GravaProcesso => "DB421_EscritaRfid".RfidEscrita[4])
   END_RUNG
   // the same network as SCL:
   "DB400_LogicaRfid"(In_ManAuto := "DB500_SinaisIhm".ManualAutomatico,   // "FB400_LogicaRfid"
                      In_LeituraEscrita := "DB1_DatabaseAgv".RFID.Inputs.Command,
                      In_Comando := "DB420_LeituraRfid".RfidLeitura[2],
                      In_OldComando := "DB3_Memorias".Rfid.Comando,
                      In_Velocidade := "DB420_LeituraRfid".RfidLeitura[3],
                      In_Linha := "DB420_LeituraRfid".RfidLeitura[4],
                      In_Posto := "DB420_LeituraRfid".RfidLeitura[1],
                      In_TagPresente := "DB1_DatabaseAgv".RFID.TagPresente,
                      In_HmiProcesso := "DB500_SinaisIhm".Processo,
                      In_GravaPosto := "DB500_SinaisIhm".PostoRfid,
                      In_GravaComando := "DB500_SinaisIhm".ComandoRfid,
                      In_GravaVel := "DB500_SinaisIhm".VelocidadeRfid,
                      In_GravaProcesso := "DB500_SinaisIhm".ProcessoRfid,
                      Out_PararAgv => "DB3_Memorias".Rfid.PararAgv,
                      Out_Comando => "DB3_Memorias".Rfid.Comando,
                      Out_Velocidade => "DB1_DatabaseAgv".RFID.Velocidade,
                      Out_Linha => "DB3_Memorias".Rfid.Linha,
                      Out_Posto => "DB3_Memorias".Rfid.Posto,
                      Out_LeituraEscrita => "DB3_Memorias".Rfid.LeituraEscrita,
                      Out_GravaPosto => "DB421_EscritaRfid".RfidEscrita[1],
                      Out_GravaComando => "DB421_EscritaRfid".RfidEscrita[2],
                      Out_GravaVel => "DB421_EscritaRfid".RfidEscrita[3],
                      Out_GravaProcesso => "DB421_EscritaRfid".RfidEscrita[4]);
END_REGION

REGION Network 3: Logica do PGV
   // Este bloco controla a logica de direção do AGV, lendo os dados do PGV e os processando por meio de um controle proporcional.
   RUNG wire#powerrail
      "DB300_LogicaPgv"(In_Emergencia := wire#w1, In_PosicaoY := "DB1_DatabaseAgv".PGV.Module2.PositionY, In_Angulo := "DB1_DatabaseAgv".PGV.Module2.Angle, In_ForaRota := "DB1_DatabaseAgv".PGV.Module2.Status.NP, In_ManAuto := "DB500_SinaisIhm".ManualAutomatico, In_Start := "DB500_SinaisIhm".Start, In_RotaEscolhida := "DB1_DatabaseAgv".PGV.Rota, Out_Angulo => "DB3_Memorias".Pgv.Angulo, Out_Direita => "DB3_Memorias".Pgv.Direita, Out_Esquerda => "DB3_Memorias".Pgv.Esquerda, Out_NaRota => "DB3_Memorias".Pgv.NaRota, Out_EmCurva => "DB3_Memorias".EmCurva, Out_EmCurvaIntermedio => "DB3_Memorias".EmCurvaIntermediario, Out_ProcessoEscolhido => "DB500_SinaisIhm".Processo)
   END_RUNG
   RUNG wire#powerrail
      I_Contact( "DB1_DatabaseAgv".Entradas.BotaoEmergencia )
   END_RUNG wire#w1
   // the same network as SCL:
   "DB300_LogicaPgv"(In_PosicaoY := "DB1_DatabaseAgv".PGV.Module2.PositionY,   // "FB300_LogicaPgv"
                     In_Angulo := "DB1_DatabaseAgv".PGV.Module2.Angle,
                     In_ForaRota := "DB1_DatabaseAgv".PGV.Module2.Status.NP,
                     In_Emergencia := NOT "DB1_DatabaseAgv".Entradas.BotaoEmergencia,
                     In_ManAuto := "DB500_SinaisIhm".ManualAutomatico,
                     In_Start := "DB500_SinaisIhm".Start,
                     In_RotaEscolhida := "DB1_DatabaseAgv".PGV.Rota,
                     Out_Angulo => "DB3_Memorias".Pgv.Angulo,
                     Out_Direita => "DB3_Memorias".Pgv.Direita,
                     Out_Esquerda => "DB3_Memorias".Pgv.Esquerda,
                     Out_NaRota => "DB3_Memorias".Pgv.NaRota,
                     Out_EmCurva => "DB3_Memorias".EmCurva,
                     Out_EmCurvaIntermedio => "DB3_Memorias".EmCurvaIntermediario,
                     Out_ProcessoEscolhido => "DB500_SinaisIhm".Processo);
END_REGION

REGION Network 4: AGV Start Stop
   // Este bloco controla o start do AGV
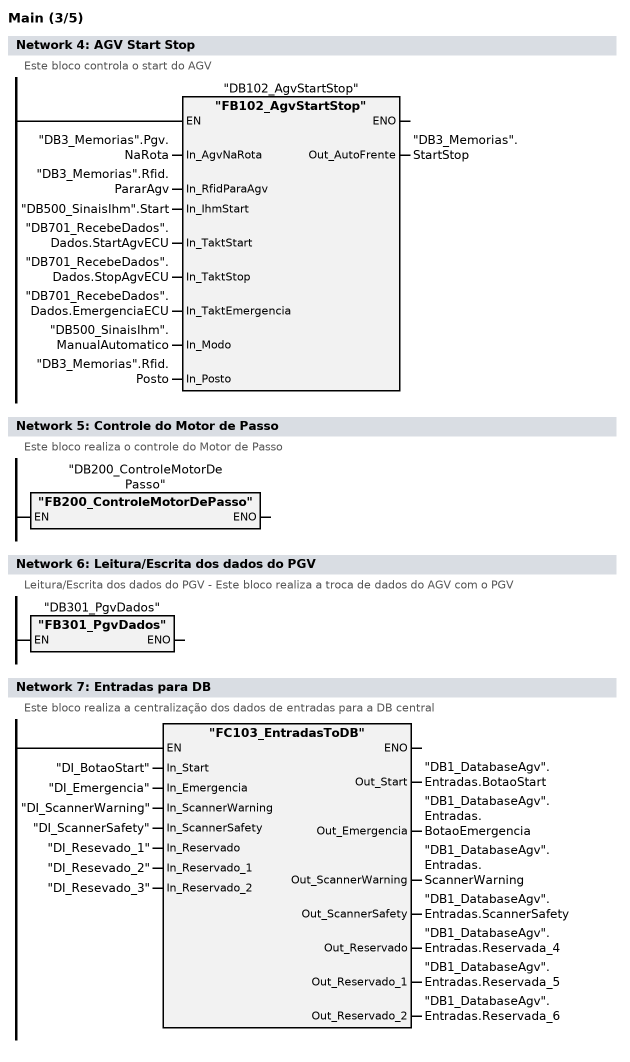
   RUNG wire#powerrail
      "DB102_AgvStartStop"(In_AgvNaRota := "DB3_Memorias".Pgv.NaRota, In_RfidParaAgv := "DB3_Memorias".Rfid.PararAgv, In_IhmStart := "DB500_SinaisIhm".Start, In_TaktStart := "DB701_RecebeDados".Dados.StartAgvECU, In_TaktStop := "DB701_RecebeDados".Dados.StopAgvECU, In_TaktEmergencia := "DB701_RecebeDados".Dados.EmergenciaECU, In_Modo := "DB500_SinaisIhm".ManualAutomatico, In_Posto := "DB3_Memorias".Rfid.Posto, Out_AutoFrente => "DB3_Memorias".StartStop)
   END_RUNG
   // the same network as SCL:
   "DB102_AgvStartStop"(In_AgvNaRota := "DB3_Memorias".Pgv.NaRota,   // "FB102_AgvStartStop"
                        In_RfidParaAgv := "DB3_Memorias".Rfid.PararAgv,
                        In_IhmStart := "DB500_SinaisIhm".Start,
                        In_TaktStart := "DB701_RecebeDados".Dados.StartAgvECU,
                        In_TaktStop := "DB701_RecebeDados".Dados.StopAgvECU,
                        In_TaktEmergencia := "DB701_RecebeDados".Dados.EmergenciaECU,
                        In_Modo := "DB500_SinaisIhm".ManualAutomatico,
                        In_Posto := "DB3_Memorias".Rfid.Posto,
                        Out_AutoFrente => "DB3_Memorias".StartStop);
END_REGION

REGION Network 5: Controle do Motor de Passo
   // Este bloco realiza o controle do Motor de Passo
   RUNG wire#powerrail
      "DB200_ControleMotorDePasso"()
   END_RUNG
   // the same network as SCL:
   "DB200_ControleMotorDePasso"();   // "FB200_ControleMotorDePasso"
END_REGION

REGION Network 6: Leitura/Escrita dos dados do PGV
   // Leitura/Escrita dos dados do PGV - Este bloco realiza a troca de dados do AGV com o PGV
   RUNG wire#powerrail
      "DB301_PgvDados"()
   END_RUNG
   // the same network as SCL:
   "DB301_PgvDados"();   // "FB301_PgvDados"
END_REGION

REGION Network 7: Entradas para DB
   // Este bloco realiza a centralização dos dados de entradas para a DB central
   RUNG wire#powerrail
      "FC103_EntradasToDB"(In_Start := "DI_BotaoStart", In_Emergencia := "DI_Emergencia", In_ScannerWarning := "DI_ScannerWarning", In_ScannerSafety := "DI_ScannerSafety", In_Reservado := "DI_Resevado_1", In_Reservado_1 := "DI_Resevado_2", In_Reservado_2 := "DI_Resevado_3", Out_Start => "DB1_DatabaseAgv".Entradas.BotaoStart, Out_Emergencia => "DB1_DatabaseAgv".Entradas.BotaoEmergencia, Out_ScannerWarning => "DB1_DatabaseAgv".Entradas.ScannerWarning, Out_ScannerSafety => "DB1_DatabaseAgv".Entradas.ScannerSafety, Out_Reservado => "DB1_DatabaseAgv".Entradas.Reservada_4, Out_Reservado_1 => "DB1_DatabaseAgv".Entradas.Reservada_5, Out_Reservado_2 => "DB1_DatabaseAgv".Entradas.Reservada_6)
   END_RUNG
   // the same network as SCL:
   "FC103_EntradasToDB"(In_Start := "DI_BotaoStart",
                        In_Emergencia := "DI_Emergencia",
                        In_ScannerWarning := "DI_ScannerWarning",
                        In_ScannerSafety := "DI_ScannerSafety",
                        In_Reservado := "DI_Resevado_1",
                        In_Reservado_1 := "DI_Resevado_2",
                        In_Reservado_2 := "DI_Resevado_3",
                        Out_Start => "DB1_DatabaseAgv".Entradas.BotaoStart,
                        Out_Emergencia => "DB1_DatabaseAgv".Entradas.BotaoEmergencia,
                        Out_ScannerWarning => "DB1_DatabaseAgv".Entradas.ScannerWarning,
                        Out_ScannerSafety => "DB1_DatabaseAgv".Entradas.ScannerSafety,
                        Out_Reservado => "DB1_DatabaseAgv".Entradas.Reservada_4,
                        Out_Reservado_1 => "DB1_DatabaseAgv".Entradas.Reservada_5,
                        Out_Reservado_2 => "DB1_DatabaseAgv".Entradas.Reservada_6);
END_REGION

REGION Network 8: DB para Saidas
   // Este bloco realiza a centralização dos dados de entradas para a DB central
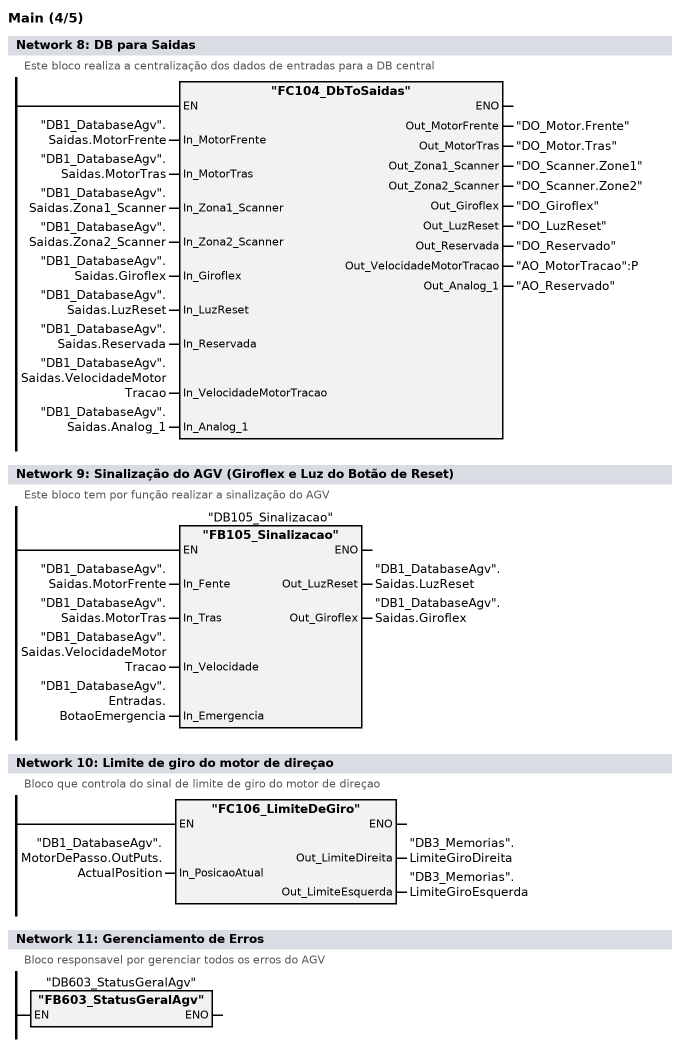
   RUNG wire#powerrail
      "FC104_DbToSaidas"(In_MotorFrente := "DB1_DatabaseAgv".Saidas.MotorFrente, In_MotorTras := "DB1_DatabaseAgv".Saidas.MotorTras, In_Zona1_Scanner := "DB1_DatabaseAgv".Saidas.Zona1_Scanner, In_Zona2_Scanner := "DB1_DatabaseAgv".Saidas.Zona2_Scanner, In_Giroflex := "DB1_DatabaseAgv".Saidas.Giroflex, In_LuzReset := "DB1_DatabaseAgv".Saidas.LuzReset, In_Reservada := "DB1_DatabaseAgv".Saidas.Reservada, In_VelocidadeMotorTracao := "DB1_DatabaseAgv".Saidas.VelocidadeMotorTracao, In_Analog_1 := "DB1_DatabaseAgv".Saidas.Analog_1, Out_MotorFrente => "DO_Motor.Frente", Out_MotorTras => "DO_Motor.Tras", Out_Zona1_Scanner => "DO_Scanner.Zone1", Out_Zona2_Scanner => "DO_Scanner.Zone2", Out_Giroflex => "DO_Giroflex", Out_LuzReset => "DO_LuzReset", Out_Reservada => "DO_Reservado", Out_VelocidadeMotorTracao => "AO_MotorTracao":P, Out_Analog_1 => "AO_Reservado")
   END_RUNG
   // the same network as SCL:
   "FC104_DbToSaidas"(In_MotorFrente := "DB1_DatabaseAgv".Saidas.MotorFrente,
                      In_MotorTras := "DB1_DatabaseAgv".Saidas.MotorTras,
                      In_Zona1_Scanner := "DB1_DatabaseAgv".Saidas.Zona1_Scanner,
                      In_Zona2_Scanner := "DB1_DatabaseAgv".Saidas.Zona2_Scanner,
                      In_Giroflex := "DB1_DatabaseAgv".Saidas.Giroflex,
                      In_LuzReset := "DB1_DatabaseAgv".Saidas.LuzReset,
                      In_Reservada := "DB1_DatabaseAgv".Saidas.Reservada,
                      In_VelocidadeMotorTracao := "DB1_DatabaseAgv".Saidas.VelocidadeMotorTracao,
                      In_Analog_1 := "DB1_DatabaseAgv".Saidas.Analog_1,
                      Out_MotorFrente => "DO_Motor.Frente",
                      Out_MotorTras => "DO_Motor.Tras",
                      Out_Zona1_Scanner => "DO_Scanner.Zone1",
                      Out_Zona2_Scanner => "DO_Scanner.Zone2",
                      Out_Giroflex => "DO_Giroflex",
                      Out_LuzReset => "DO_LuzReset",
                      Out_Reservada => "DO_Reservado",
                      Out_VelocidadeMotorTracao => "AO_MotorTracao":P,
                      Out_Analog_1 => "AO_Reservado");
END_REGION

REGION Network 9: Sinalização do AGV (Giroflex e Luz do Botão de Reset)
   // Este bloco tem por função realizar a sinalização do AGV
   RUNG wire#powerrail
      "DB105_Sinalizacao"(In_Fente := "DB1_DatabaseAgv".Saidas.MotorFrente, In_Tras := "DB1_DatabaseAgv".Saidas.MotorTras, In_Velocidade := "DB1_DatabaseAgv".Saidas.VelocidadeMotorTracao, In_Emergencia := "DB1_DatabaseAgv".Entradas.BotaoEmergencia, Out_LuzReset => "DB1_DatabaseAgv".Saidas.LuzReset, Out_Giroflex => "DB1_DatabaseAgv".Saidas.Giroflex)
   END_RUNG
   // the same network as SCL:
   "DB105_Sinalizacao"(In_Fente := "DB1_DatabaseAgv".Saidas.MotorFrente,   // "FB105_Sinalizacao"
                       In_Tras := "DB1_DatabaseAgv".Saidas.MotorTras,
                       In_Velocidade := "DB1_DatabaseAgv".Saidas.VelocidadeMotorTracao,
                       In_Emergencia := "DB1_DatabaseAgv".Entradas.BotaoEmergencia,
                       Out_LuzReset => "DB1_DatabaseAgv".Saidas.LuzReset,
                       Out_Giroflex => "DB1_DatabaseAgv".Saidas.Giroflex);
END_REGION

REGION Network 10: Limite de giro do motor de direçao
   // Bloco que controla do sinal de limite de giro do motor de direçao
   RUNG wire#powerrail
      "FC106_LimiteDeGiro"(In_PosicaoAtual := "DB1_DatabaseAgv".MotorDePasso.OutPuts.ActualPosition, Out_LimiteDireita => "DB3_Memorias".LimiteGiroDireita, Out_LimiteEsquerda => "DB3_Memorias".LimiteGiroEsquerda)
   END_RUNG
   // the same network as SCL:
   "FC106_LimiteDeGiro"(In_PosicaoAtual := "DB1_DatabaseAgv".MotorDePasso.OutPuts.ActualPosition,
                        Out_LimiteDireita => "DB3_Memorias".LimiteGiroDireita,
                        Out_LimiteEsquerda => "DB3_Memorias".LimiteGiroEsquerda);
END_REGION

REGION Network 11: Gerenciamento de Erros
   // Bloco responsavel por gerenciar todos os erros do AGV
   RUNG wire#powerrail
      "DB603_StatusGeralAgv"()
   END_RUNG
   // the same network as SCL:
   "DB603_StatusGeralAgv"();   // "FB603_StatusGeralAgv"
END_REGION

REGION Network 12: Comunicação com o Takt
   // Realiza a comunicação com o takt (Leitura e escrita)
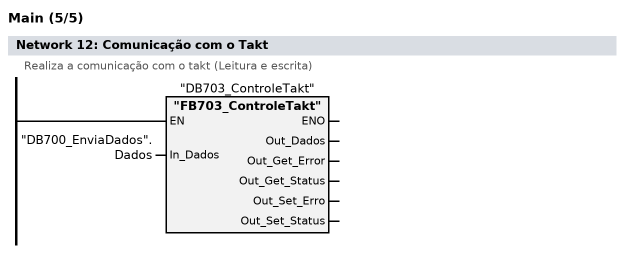
   RUNG wire#powerrail
      "DB703_ControleTakt"(In_Dados := "DB700_EnviaDados".Dados, Out_Dados =>, Out_Get_Error =>, Out_Get_Status =>, Out_Set_Erro =>, Out_Set_Status =>)
   END_RUNG
   // the same network as SCL:
   "DB703_ControleTakt"(In_Dados := "DB700_EnviaDados".Dados);   // "FB703_ControleTakt"
END_REGION
END_ORGANIZATION_BLOCK

// folder: 01_Controle/01_Function

FUNCTION_BLOCK "FB100_ManualAutomatico"   // FB1, SCL
TITLE = FB100_ManualAutomatico
{ S7_Optimized_Access := 'FALSE' }
AUTHOR : ssbjvq
FAMILY : AGV_KD
VERSION : 1.0
// Este bloco é responsavel por realizar o controle do AGV no modo automatico e no modo manual, sem ele o AGV não realiza nenhum movimento.
   VAR_INPUT
      In_ManFrente : Bool;   // Sinal de comando manual no sentido frente, vindo da IHM
      In_ManTras : Bool;   // Sinal de comando manual no sentido tras, vindo da IHM
      In_ManEsquerda : Bool;   // Sinal de comando manual no sentido esquerda, vindo da IHM
      In_ManDireita : Bool;   // Sinal de comando manual no sentido direita, vindo da IHM
      In_Emergencia : Bool;   // Sinal de emergencia do AGV
      In_AutoFrente : Bool;   // Sinal de comando automatico no sentido frente, vindo da logica do CLP externa.
      In_AutoEsquerda : Bool;   // Sinal de comando automatico no sentido esquerda, vindo do bloco do PGV.
      In_AutoDireita : Bool;   // Sinal de comando automatico no sentido direita, vindo do bloco do PGV.
      In_Safety : Bool;   // Sinal de area de segurança do Scanner de seguraça acionada
      In_Warning : Bool;   // Sinal de area de atenção do Scanner de seguraça acionada
      In_ManVel : Int;   // Valor de velocidade do AGV no modo manual, vindo da IHM.
      In_AutoVel : Int;   // Valor de velocidade do AGV no modo automatico, vindo do controle do Rfid.
      In_AutoWarning : Int;   // Valor de velocidade do AGV no modo manual, vindo da logica do CLP.
      In_ManAuto : Int;   // Memoria que escolhe o modo de operação, se é automatico/manual.
      In_Start : Bool;   // Memoria de start do AGV
      In_EmCurva : Bool;   // Sinal que indica que o AGV esta em curva fechada, vindo do bloco do PGV
      In_NaRota : Bool;   // Sinal que indica que o AGV esta na rota, vindo do bloco do PGV
      In_EmCurvaIntermediario : Bool;   // Sinal que indica que o AGV esta em curva, vindo do bloco do PGV
      In_ActualPosition : DInt;   // Sinal que mostra a atual posição do motor de passo
   END_VAR
   VAR_OUTPUT
      Out_Frente : Bool;   // Sinal de sentido de giro do motor do AGV para frente
      Out_Tras : Bool;   // Sinal de sentido de giro do motor do AGV para tras
      Out_Esquerda : Bool;   // Sinal de sentido do AGV para esquerda
      Out_Direita : Bool;   // Sinal de sentido do AGV para direita
      Out_Posicao : DInt;   // Sinal de posição atual do motor de passo
      Out_Velocidade : Int;   // Sinal que controla a velocidade do motor de tração
   END_VAR
   VAR
      TOF_MotorTras : TOF;   // Temporizador utilizado para o gerar o delay quando o comando da ihm de manual frente for desacionado.
      TOF_MotorAutomatico : TOF;   // Temporizador utilizado para o gerar o delay quando o comando da ihm de manual tras for desacionado.
      TOF_MotorFrente : TOF;   // Temporizador utilizado para o gerar o delay no modo automatico.
      S_Frente : Bool;   // Memoria Frente
      S_Tras : Bool;   // Memoria Tras
      S_Esquerda : Bool;   // Memoria esquerda
      S_Direita : Bool;   // Memoria direita
      ControleVelocidade : "FB101_ControleVelocidade";   // Bloco que realiza o controle de acelaração e desaceleração do motor de tração
      S_Vel : Int;   // Valor de velocidade inputado no bloco de controle de velocidade
      S_AutoVel : Int;   // Velocida em automatico
      S_AutoWarning : Int;   // Valor velocidade em warning
      S_VelMan : Int;   // Valor velocidade em manual
   END_VAR
BEGIN
   (*
   Este bloco é responsavel por realizar o controle do AGV no modo automatico e no modo manual, sem ele o AGV não realiza nenhum movimento.
   *)

   // Delay de parada do motor.
   REGION Temporizadores
       (*
         - Estes temporizadores, são os responsaveis por gerar um delay para controlar e realizar a parada gradual/desaceleração do AGV.
         - Um temporizador para cada movimento.
       *) 

       //Temporizador utilizado para o gerar o delay quando o comando da ihm de manual frente for desacionado.
       #TOF_MotorFrente(IN := #In_ManFrente,
                        PT := T#1.5s);
       //Temporizador utilizado para o gerar o delay quando o comando da ihm de manual tras for desacionado.
       #TOF_MotorTras(IN := #In_ManTras,
                      PT := T#1.5s);
       //Temporizador utilizado para o gerar o delay no modo automatico.
       #TOF_MotorAutomatico(IN := ((#In_AutoFrente AND #In_Start AND NOT #In_NaRota) OR (#In_AutoFrente AND #In_Start)),
                            PT := T#1.8s);
   END_REGION

   // Coloca os parametros de velocidade em uma memoria.
   REGION MemoriasVelocidades    
       // Coloca os parametros de velocidade em uma memoria e em alguns casos realiza uma conta.
       #S_AutoVel := #In_AutoVel;
       #S_AutoWarning := #In_AutoWarning * 1000;
       #S_VelMan := #In_ManVel;

   END_REGION

   //Logica central do bloco
   REGION ContorleDosAcionamentos
       //Verificação se o emergencia não esta acionado
       IF #In_Emergencia THEN
           // Se estiver em modo manual envia os comando e a velocidade
           IF #In_ManAuto = 1 AND NOT #TOF_MotorAutomatico.Q THEN
               IF (#In_ManFrente OR #TOF_MotorFrente.Q) AND NOT #In_ManTras THEN
                   #S_Frente := 1;
                   #S_Tras := 0;
                   #S_Vel := #S_VelMan;
               ELSIF (#In_ManTras OR #TOF_MotorTras.Q) AND NOT #In_ManFrente THEN
                   #S_Tras := 1;
                   #S_Frente := 0;
                   #S_Vel := #S_VelMan;
               ELSE
                   #S_Frente := 0;
                   #S_Tras := 0;
               END_IF;
               // Controla o motor de direção
               IF #In_ManEsquerda AND NOT #In_ManDireita AND (#In_ActualPosition < 6000) THEN
                   #S_Esquerda := 1;
               ELSIF #In_ManDireita AND NOT #In_ManEsquerda AND (#In_ActualPosition > -6000) THEN
                   #S_Direita := 1;
               ELSE
                   #S_Esquerda := 0;
                   #S_Direita := 0;
               END_IF;


               // Se estiver em modo Automatico
           ELSIF #In_ManAuto = 2 OR #TOF_MotorAutomatico.Q THEN

               #S_Vel := #S_AutoVel;
               // Controla o motor de direção
               IF (#In_ActualPosition < 6000) THEN
                   #S_Esquerda := #In_AutoEsquerda;
               ELSE
                   #S_Esquerda := 0;
               END_IF;
               // Controla o motor de direção
               IF (#In_ActualPosition > -6000) THEN
                   #S_Direita := #In_AutoDireita;
               ELSE
                   #S_Direita := 0;
               END_IF;

               //Libera o bloco de controle de velocida á enviar velocidade
               #S_Frente := (#In_AutoFrente AND #In_Start AND #In_NaRota) OR #TOF_MotorAutomatico.Q;
           ELSE
               #S_Esquerda := 0;
               #S_Direita := 0;
               #S_Frente := 0;
               #S_Tras := 0;
           END_IF;
       ELSE
           #S_Esquerda := 0;
           #S_Direita := 0;
           #S_Frente := 0;
           #S_Tras := 0;
       END_IF;
   END_REGION

   //Realiza o controle da velocidade
   REGION BlocoDeControleDeVelocidade
       #ControleVelocidade(In_ManFrente := #In_ManFrente,
                           In_ManTras := #In_ManTras,
                           In_AutoFrente := (#In_AutoFrente AND #In_Start),
                           In_Emergencia := NOT #In_Emergencia,
                           In_Safety := #In_Safety,
                           In_Warning := #In_Warning,
                           In_Vel := #S_Vel,
                           In_ManAuto := #In_ManAuto,
                           In_VelWarning := #In_AutoWarning,
                           In_VelIntermediario := 14,
                           In_NaRota := #In_NaRota,
                           In_EmCurvaIntermediario := #In_EmCurvaIntermediario,
                           In_EmCurva := #In_EmCurva,
                           Out_Velocidade => #Out_Velocidade);
   END_REGION

   REGION Outputs
       //Coloca os valores das memorias nas saidas
       #Out_Esquerda := #S_Esquerda;
       #Out_Direita := #S_Direita;
       #Out_Frente := #S_Frente;
       #Out_Tras := #S_Tras;
   END_REGION
END_FUNCTION_BLOCK

FUNCTION_BLOCK "FB101_ControleVelocidade"   // FB2, SCL
TITLE = FB101_ControleVelocidade
{ S7_Optimized_Access := 'FALSE' }
AUTHOR : ssbjvq
FAMILY : AGV_KD
VERSION : 1.0
// Bloco que realiza o controle de acelaração e desaceleração do motor de tração
   VAR_INPUT
      In_ManFrente : Bool;   // Sinal de comando manual no sentido frente, vindo da IHM
      In_ManTras : Bool;   // Sinal de comando manual no sentido tras, vindo da IHM
      In_AutoFrente : Bool;   // Sinal de acionamento do automatico frente
      In_Emergencia : Bool;   // Sinal de emergencia do AGV
      In_Safety : Bool;   // Sinal de area de segurança do Scanner de seguraça acionada
      In_Warning : Bool;   // Sinal de area de atenção do Scanner de seguraça acionada
      In_Vel : Int;   // Valor de velocidade do AGV
      In_ManAuto : Int;   // Memoria que escolhe o modo de operação, se é automatico/manual.
      In_VelWarning : Int;   // Sinal de velocidade em modo atenção do Scanner
      In_VelIntermediario : Int;   // Sinal de velocidade em modo de curva intermediaria
      In_NaRota : Bool;   // Sinal se o agv esta na rota
      In_EmCurvaIntermediario : Bool;   // Sinal de curva intermediaria
      In_EmCurva : Bool;   // Sinal de curva
   END_VAR
   VAR_OUTPUT
      Out_Velocidade : Int;   // Sinal de saida na velocidade do AGV
   END_VAR
   VAR
      S_AuxVel : Int;   // Memoria de valor de velocidade
   END_VAR
BEGIN
   (*
       Bloco que realiza o controle de acelaração e desaceleração do motor de tração
   *)


   //Cria o limite de velocidade
   REGION LimiteDeVelocidade
       //Limita a velocidade de 27000 inteiros a 10000 inteiros
       IF #In_Vel > 27 THEN
           #S_AuxVel := 27000;
       ELSIF #In_Vel < 0 THEN
           #S_AuxVel := 10000;
       ELSE
           #S_AuxVel := #In_Vel * 1000;
       END_IF;
   END_REGION

   //Controla o envio de velocidade para o motor
   REGION LogicaDeControle

       //Se o emergencia estiver acionado ou o a area de segurança do scanner em modo automatico
       IF #In_Emergencia OR (#In_Safety AND #In_ManAuto <> 1) THEN
           #Out_Velocidade := 0;
       //Senão se as memorias de movimento estiver aciona    
       ELSIF #In_ManFrente OR #In_ManTras OR #In_AutoFrente THEN

           // Reduz a velocidade em curva intermediaria para o valor especificado
           IF #In_EmCurvaIntermediario AND NOT #In_EmCurva
               AND #Out_Velocidade >= (#In_VelIntermediario * 1000)
               AND (#In_ManAuto = 2) THEN

               #Out_Velocidade := #Out_Velocidade - 150;

               // Reduz a velocidade em curva/Warning scanner para o valor especificado
           ELSIF NOT #In_EmCurvaIntermediario AND (#In_EmCurva OR #In_Warning)
               AND #Out_Velocidade >= (#In_VelWarning * 1000)
               AND (#In_ManAuto = 2) THEN

               #Out_Velocidade := #Out_Velocidade - 50;

           ELSE
               // Controle de aceleração
               IF #Out_Velocidade >= #S_AuxVel THEN
                   #Out_Velocidade := #S_AuxVel;
               ELSE
                   #Out_Velocidade := #Out_Velocidade + 10;
               END_IF;
           END_IF;

           // Controle de desaceleração
       ELSIF (NOT #In_ManFrente OR NOT #In_ManTras OR NOT #In_AutoFrente) AND #Out_Velocidade > 0 THEN
           #Out_Velocidade := #Out_Velocidade - 10;//25

           //Controla para não ter valor de velocidade negativo
           IF #Out_Velocidade < 3 THEN
               #Out_Velocidade := 0;
               ;
           END_IF;

       END_IF;

   END_REGION
END_FUNCTION_BLOCK

FUNCTION_BLOCK "FB102_AgvStartStop"   // FB3, LAD
TITLE = Este bloco controla o start do AGV
{ S7_Optimized_Access := 'FALSE' }
VERSION : 0.1
// Este bloco controla o start do AGV
   VAR_INPUT
      In_AgvNaRota : Bool;   // Sinal de AGV na rota, vindo do bloco do PGV
      In_RfidParaAgv : Bool;   // Sinal de parada do AGV por conta da Tag RFID
      In_IhmStart : Bool;   // Sinal de start do AGV pela IHM
      In_TaktStart : Bool;   // Sinal de start do AGV pelo TAKT
      In_TaktStop : Bool;   // Sinal de stop do AGV pelo TAKT
      In_TaktEmergencia : Bool;   // Sinal de Emergencia acionado de algum dispositivo, vindo da comunicação com o takt
      In_Modo : Int;   // Sinal do modo aut/man
      In_Posto : Int;   // Sinal Sinal do posto em que o AGV esta
   END_VAR
   VAR_OUTPUT
      Out_AutoFrente : Bool;   // Acionamento do start do AGV em moto automatico
   END_VAR
   VAR
      TON_NaRota : TON;   // Temporizador de fora da rota
      Pulse_Rfid : Bool;   // Memoria de pulso do sinal de para AGV
   END_VAR
   VAR_TEMP   // added for the SCL form of the ladder/FBD networks
      _w1 : Bool;
   END_VAR
BEGIN

REGION Network 1: Set Memoria
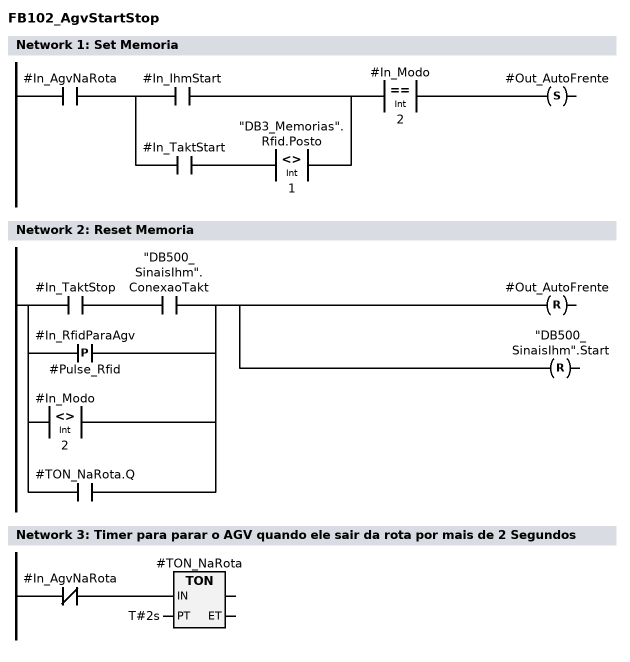
   RUNG wire#powerrail
      Contact( #In_AgvNaRota )
      wire#w1
      Contact( #In_IhmStart )
      wire#w2
      { S7_Templates := "SrcType := Int" } EQ_Contact(in1 := #In_Modo, in2 := 2)
      S_Coil( #Out_AutoFrente )
   END_RUNG
   RUNG wire#w1
      Contact( #In_TaktStart )
      { S7_Templates := "SrcType := Int" } NE_Contact(in1 := "DB3_Memorias".Rfid.Posto, in2 := 1)
   END_RUNG wire#w2
   // the same network as SCL:
   IF #In_AgvNaRota AND (#In_IhmStart OR (#In_TaktStart AND ("DB3_Memorias".Rfid.Posto <> 1))) AND (#In_Modo = 2) THEN
       #Out_AutoFrente := TRUE;
   END_IF;
END_REGION

REGION Network 2: Reset Memoria
   RUNG wire#powerrail
      Contact( #In_TaktStop )
      Contact( "DB500_SinaisIhm".ConexaoTakt )
      wire#w1
      R_Coil( #Out_AutoFrente )
   END_RUNG
   RUNG wire#powerrail
      P_Contact(operand := #In_RfidParaAgv, bit := #Pulse_Rfid)
   END_RUNG wire#w1
   RUNG wire#powerrail
      { S7_Templates := "SrcType := Int" } NE_Contact(in1 := #In_Modo, in2 := 2)
   END_RUNG wire#w1
   RUNG wire#powerrail
      Contact( #TON_NaRota.Q )
   END_RUNG wire#w1
   RUNG wire#w1
      R_Coil( "DB500_SinaisIhm".Start )
   END_RUNG
   // the same network as SCL:
   #_w1 := #In_RfidParaAgv AND NOT #Pulse_Rfid;   // rising edge of #In_RfidParaAgv
   #Pulse_Rfid := #In_RfidParaAgv;
   IF (#In_TaktStop AND "DB500_SinaisIhm".ConexaoTakt) OR #_w1 OR (#In_Modo <> 2) OR #TON_NaRota.Q THEN
       #Out_AutoFrente := FALSE;
       "DB500_SinaisIhm".Start := FALSE;
   END_IF;
END_REGION

REGION Network 3: Timer para parar o AGV quando ele sair da rota por mais de 2 Segundos
   #TON_NaRota.TON(IN := NOT #In_AgvNaRota, PT := T#2s);
END_REGION
END_FUNCTION_BLOCK

FUNCTION_BLOCK "FB105_Sinalizacao"   // FB105, SCL
TITLE = FB105_Sinalizacao
{ S7_Optimized_Access := 'FALSE' }
AUTHOR : ssbjvq
FAMILY : AGV_KD
VERSION : 0.1
// Este bloco tem por função realizar a sinalização do AGV
   VAR_INPUT
      In_Fente : Bool;
      In_Tras : Bool;
      In_Velocidade : Int;
      In_Emergencia : Bool;
   END_VAR
   VAR_OUTPUT
      Out_LuzReset : Bool;
      Out_Giroflex : Bool;
   END_VAR
BEGIN


   IF (#In_Fente OR #In_Tras) AND #In_Velocidade > 0 THEN
       #Out_Giroflex := 1;
   ELSE
       #Out_Giroflex := 0;
   END_IF;

   IF #In_Emergencia THEN
       #Out_LuzReset := 1;
   ELSE
       #Out_LuzReset := 0;
   END_IF;
END_FUNCTION_BLOCK

FUNCTION "FC103_EntradasToDB" : Void   // FC103, SCL
TITLE = FC103_EntradasToDB
{ S7_Optimized_Access := 'FALSE' }
AUTHOR : ssbjvq
FAMILY : AGV_KD
VERSION : 0.1
// Este bloco realiza a centralização dos dados de entradas para a DB central
   VAR_INPUT
      In_Start : Bool;
      In_Emergencia : Bool;
      In_ScannerWarning : Bool;
      In_ScannerSafety : Bool;
      In_Reservado : Bool;
      In_Reservado_1 : Bool;
      In_Reservado_2 : Bool;
   END_VAR
   VAR_OUTPUT
      Out_Start : Bool;
      Out_Emergencia : Bool;
      Out_ScannerWarning : Bool;
      Out_ScannerSafety : Bool;
      Out_Reservado : Bool;
      Out_Reservado_1 : Bool;
      Out_Reservado_2 : Bool;
   END_VAR
BEGIN



   #Out_Start := #In_Start;
   #Out_Emergencia := #In_Emergencia;
   #Out_ScannerWarning := #In_ScannerWarning;
   #Out_ScannerSafety := #In_ScannerSafety;
   #Out_Reservado := #In_Reservado;
   #Out_Reservado_1 := #In_Reservado_1;
   #Out_Reservado_2 := #In_Reservado_2;
END_FUNCTION

FUNCTION "FC104_DbToSaidas" : Void   // FC104, SCL
TITLE = FC104_DbToSaidas
{ S7_Optimized_Access := 'FALSE' }
AUTHOR : ssbjvq
FAMILY : AGV_KD
VERSION : 0.1
// Este bloco realiza a centralização dos dados de entradas para a DB central
   VAR_INPUT
      In_MotorFrente : Bool;
      In_MotorTras : Bool;
      In_Zona1_Scanner : Bool;
      In_Zona2_Scanner : Bool;
      In_Giroflex : Bool;
      In_LuzReset : Bool;
      In_Reservada : Bool;
      In_VelocidadeMotorTracao : Int;
      In_Analog_1 : Int;
   END_VAR
   VAR_OUTPUT
      Out_MotorFrente : Bool;
      Out_MotorTras : Bool;
      Out_Zona1_Scanner : Bool;
      Out_Zona2_Scanner : Bool;
      Out_Giroflex : Bool;
      Out_LuzReset : Bool;
      Out_Reservada : Bool;
      Out_VelocidadeMotorTracao : Int;
      Out_Analog_1 : Int;
   END_VAR
BEGIN
   #Out_MotorFrente := #In_MotorFrente;
   #Out_MotorTras := #In_MotorTras;
   #Out_Zona1_Scanner := #In_Zona1_Scanner;
   #Out_Zona2_Scanner := #In_Zona2_Scanner;
   #Out_Giroflex := #In_Giroflex;
   #Out_LuzReset := #In_LuzReset;
   #Out_Reservada := #In_Reservada;
   #Out_VelocidadeMotorTracao := #In_VelocidadeMotorTracao;
   #Out_Analog_1 := #In_Analog_1;
END_FUNCTION

FUNCTION "FC106_LimiteDeGiro" : Void   // FC106, SCL
TITLE = FC106_LimiteDeGiro
{ S7_Optimized_Access := 'FALSE' }
AUTHOR : ssbjvq
FAMILY : AGV_KD
VERSION : 0.1
// Bloco que controla do sinal de limite de giro do motor de direçao
   VAR_INPUT
      In_PosicaoAtual : DInt;
   END_VAR
   VAR_OUTPUT
      Out_LimiteDireita : Bool;
      Out_LimiteEsquerda : Bool;
   END_VAR
BEGIN


   IF #In_PosicaoAtual >= 6000 THEN
       #Out_LimiteDireita := 0;
       #Out_LimiteEsquerda := 1;
   ELSE
       #Out_LimiteEsquerda := 0;
   END_IF;


   IF #In_PosicaoAtual <= -6000 THEN
       #Out_LimiteDireita := 1;
       #Out_LimiteEsquerda := 0;
   ELSE
       #Out_LimiteDireita := 0;
   END_IF;
END_FUNCTION

// folder: 02_MotorPasso/01_Function

FUNCTION_BLOCK "FB200_ControleMotorDePasso"   // FB200, LAD
TITLE = FB200_ControleMotorDePasso
{ S7_Optimized_Access := 'FALSE' }
AUTHOR : ssbjvq
FAMILY : AGV_KD
VERSION : 0.1
// Este bloco reune todos os blocos para o controle do motor de passo
   VAR
      FHPP_GETIO_PART_Instance : "FB203_FHPP_GETIO_PART";   // Este bloco server para realizar a leitura dos dados do motor de direção
      FHPP_CTRL_Instance : "FB204_FHPP_CTRL";   // Este é o bloco utilizado para controlar os comando e ler os status do motor
      FHPP_SETIO_PART : "FB205_FHPP_SETIO_PART";   // Este bloco server para realizar a escrita dos dados no motor de direção
      FML_REF : "DT_FML_REF";
   END_VAR
BEGIN

REGION Network 1: GET Dados Motor direção
   // Este bloco server para realizar a leitura dos dados do motor de direção
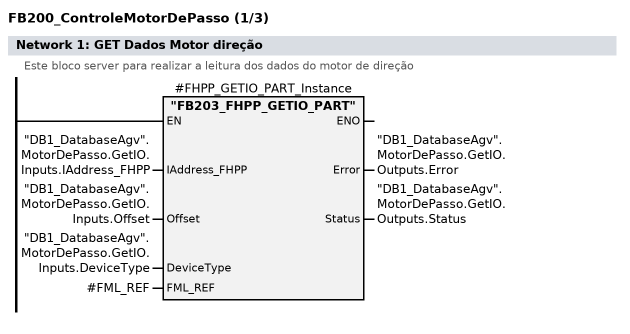
   RUNG wire#powerrail
      #FHPP_GETIO_PART_Instance(IAddress_FHPP := "DB1_DatabaseAgv".MotorDePasso.GetIO.Inputs.IAddress_FHPP, Offset := "DB1_DatabaseAgv".MotorDePasso.GetIO.Inputs.Offset, DeviceType := "DB1_DatabaseAgv".MotorDePasso.GetIO.Inputs.DeviceType, FML_REF := #FML_REF, Error => "DB1_DatabaseAgv".MotorDePasso.GetIO.Outputs.Error, Status => "DB1_DatabaseAgv".MotorDePasso.GetIO.Outputs.Status)
   END_RUNG
   // the same network as SCL:
   #FHPP_GETIO_PART_Instance(IAddress_FHPP := "DB1_DatabaseAgv".MotorDePasso.GetIO.Inputs.IAddress_FHPP,   // "FB203_FHPP_GETIO_PART"
                           Offset := "DB1_DatabaseAgv".MotorDePasso.GetIO.Inputs.Offset,
                           DeviceType := "DB1_DatabaseAgv".MotorDePasso.GetIO.Inputs.DeviceType,
                           FML_REF := #FML_REF,
                           Error => "DB1_DatabaseAgv".MotorDePasso.GetIO.Outputs.Error,
                           Status => "DB1_DatabaseAgv".MotorDePasso.GetIO.Outputs.Status);
END_REGION

REGION Network 2: Controle motor direção
   // Este é o bloco utilizado para controlar os comando e ler os status do motor
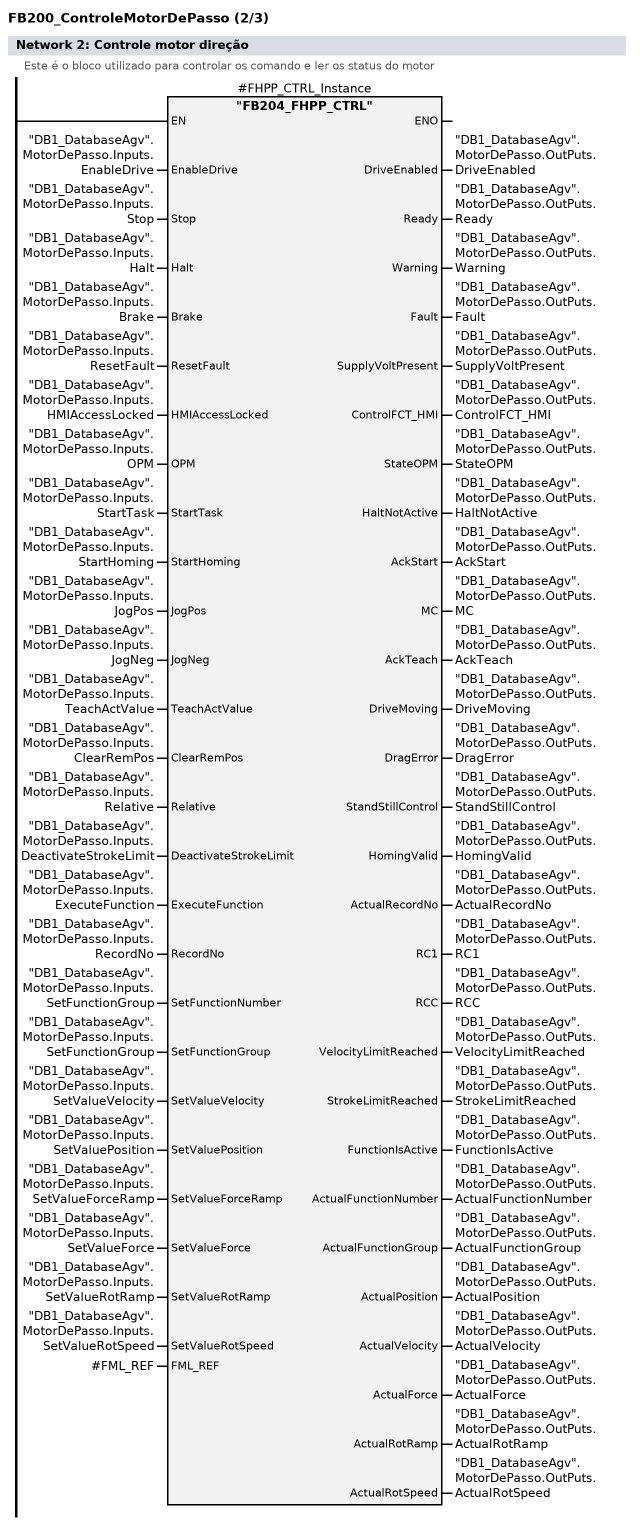
   RUNG wire#powerrail
      #FHPP_CTRL_Instance(EnableDrive := "DB1_DatabaseAgv".MotorDePasso.Inputs.EnableDrive, Stop := "DB1_DatabaseAgv".MotorDePasso.Inputs.Stop, Halt := "DB1_DatabaseAgv".MotorDePasso.Inputs.Halt, Brake := "DB1_DatabaseAgv".MotorDePasso.Inputs.Brake, ResetFault := "DB1_DatabaseAgv".MotorDePasso.Inputs.ResetFault, HMIAccessLocked := "DB1_DatabaseAgv".MotorDePasso.Inputs.HMIAccessLocked, OPM := "DB1_DatabaseAgv".MotorDePasso.Inputs.OPM, StartTask := "DB1_DatabaseAgv".MotorDePasso.Inputs.StartTask, StartHoming := "DB1_DatabaseAgv".MotorDePasso.Inputs.StartHoming, JogPos := "DB1_DatabaseAgv".MotorDePasso.Inputs.JogPos, JogNeg := "DB1_DatabaseAgv".MotorDePasso.Inputs.JogNeg, TeachActValue := "DB1_DatabaseAgv".MotorDePasso.Inputs.TeachActValue, ClearRemPos := "DB1_DatabaseAgv".MotorDePasso.Inputs.ClearRemPos, Relative := "DB1_DatabaseAgv".MotorDePasso.Inputs.Relative, DeactivateStrokeLimit := "DB1_DatabaseAgv".MotorDePasso.Inputs.DeactivateStrokeLimit, ExecuteFunction := "DB1_DatabaseAgv".MotorDePasso.Inputs.ExecuteFunction, RecordNo := "DB1_DatabaseAgv".MotorDePasso.Inputs.RecordNo, SetFunctionNumber := "DB1_DatabaseAgv".MotorDePasso.Inputs.SetFunctionGroup, SetFunctionGroup := "DB1_DatabaseAgv".MotorDePasso.Inputs.SetFunctionGroup, SetValueVelocity := "DB1_DatabaseAgv".MotorDePasso.Inputs.SetValueVelocity, SetValuePosition := "DB1_DatabaseAgv".MotorDePasso.Inputs.SetValuePosition, SetValueForceRamp := "DB1_DatabaseAgv".MotorDePasso.Inputs.SetValueForceRamp, SetValueForce := "DB1_DatabaseAgv".MotorDePasso.Inputs.SetValueForce, SetValueRotRamp := "DB1_DatabaseAgv".MotorDePasso.Inputs.SetValueRotRamp, SetValueRotSpeed := "DB1_DatabaseAgv".MotorDePasso.Inputs.SetValueRotSpeed, FML_REF := #FML_REF, DriveEnabled => "DB1_DatabaseAgv".MotorDePasso.OutPuts.DriveEnabled, Ready => "DB1_DatabaseAgv".MotorDePasso.OutPuts.Ready, Warning => "DB1_DatabaseAgv".MotorDePasso.OutPuts.Warning, Fault => "DB1_DatabaseAgv".MotorDePasso.OutPuts.Fault, SupplyVoltPresent => "DB1_DatabaseAgv".MotorDePasso.OutPuts.SupplyVoltPresent, ControlFCT_HMI => "DB1_DatabaseAgv".MotorDePasso.OutPuts.ControlFCT_HMI, StateOPM => "DB1_DatabaseAgv".MotorDePasso.OutPuts.StateOPM, HaltNotActive => "DB1_DatabaseAgv".MotorDePasso.OutPuts.HaltNotActive, AckStart => "DB1_DatabaseAgv".MotorDePasso.OutPuts.AckStart, MC => "DB1_DatabaseAgv".MotorDePasso.OutPuts.MC, AckTeach => "DB1_DatabaseAgv".MotorDePasso.OutPuts.AckTeach, DriveMoving => "DB1_DatabaseAgv".MotorDePasso.OutPuts.DriveMoving, DragError => "DB1_DatabaseAgv".MotorDePasso.OutPuts.DragError, StandStillControl => "DB1_DatabaseAgv".MotorDePasso.OutPuts.StandStillControl, HomingValid => "DB1_DatabaseAgv".MotorDePasso.OutPuts.HomingValid, ActualRecordNo => "DB1_DatabaseAgv".MotorDePasso.OutPuts.ActualRecordNo, RC1 => "DB1_DatabaseAgv".MotorDePasso.OutPuts.RC1, RCC => "DB1_DatabaseAgv".MotorDePasso.OutPuts.RCC, VelocityLimitReached => "DB1_DatabaseAgv".MotorDePasso.OutPuts.VelocityLimitReached, StrokeLimitReached => "DB1_DatabaseAgv".MotorDePasso.OutPuts.StrokeLimitReached, FunctionIsActive => "DB1_DatabaseAgv".MotorDePasso.OutPuts.FunctionIsActive, ActualFunctionNumber => "DB1_DatabaseAgv".MotorDePasso.OutPuts.ActualFunctionNumber, ActualFunctionGroup => "DB1_DatabaseAgv".MotorDePasso.OutPuts.ActualFunctionGroup, ActualPosition => "DB1_DatabaseAgv".MotorDePasso.OutPuts.ActualPosition, ActualVelocity => "DB1_DatabaseAgv".MotorDePasso.OutPuts.ActualVelocity, ActualForce => "DB1_DatabaseAgv".MotorDePasso.OutPuts.ActualForce, ActualRotRamp => "DB1_DatabaseAgv".MotorDePasso.OutPuts.ActualRotRamp, ActualRotSpeed => "DB1_DatabaseAgv".MotorDePasso.OutPuts.ActualRotSpeed)
   END_RUNG
   // the same network as SCL:
   #FHPP_CTRL_Instance(EnableDrive := "DB1_DatabaseAgv".MotorDePasso.Inputs.EnableDrive,   // "FB204_FHPP_CTRL"
                       Stop := "DB1_DatabaseAgv".MotorDePasso.Inputs.Stop,
                       Halt := "DB1_DatabaseAgv".MotorDePasso.Inputs.Halt,
                       Brake := "DB1_DatabaseAgv".MotorDePasso.Inputs.Brake,
                       ResetFault := "DB1_DatabaseAgv".MotorDePasso.Inputs.ResetFault,
                       HMIAccessLocked := "DB1_DatabaseAgv".MotorDePasso.Inputs.HMIAccessLocked,
                       OPM := "DB1_DatabaseAgv".MotorDePasso.Inputs.OPM,
                       StartTask := "DB1_DatabaseAgv".MotorDePasso.Inputs.StartTask,
                       StartHoming := "DB1_DatabaseAgv".MotorDePasso.Inputs.StartHoming,
                       JogPos := "DB1_DatabaseAgv".MotorDePasso.Inputs.JogPos,
                       JogNeg := "DB1_DatabaseAgv".MotorDePasso.Inputs.JogNeg,
                       TeachActValue := "DB1_DatabaseAgv".MotorDePasso.Inputs.TeachActValue,
                       ClearRemPos := "DB1_DatabaseAgv".MotorDePasso.Inputs.ClearRemPos,
                       Relative := "DB1_DatabaseAgv".MotorDePasso.Inputs.Relative,
                       DeactivateStrokeLimit := "DB1_DatabaseAgv".MotorDePasso.Inputs.DeactivateStrokeLimit,
                       ExecuteFunction := "DB1_DatabaseAgv".MotorDePasso.Inputs.ExecuteFunction,
                       RecordNo := "DB1_DatabaseAgv".MotorDePasso.Inputs.RecordNo,
                       SetFunctionNumber := "DB1_DatabaseAgv".MotorDePasso.Inputs.SetFunctionGroup,
                       SetFunctionGroup := "DB1_DatabaseAgv".MotorDePasso.Inputs.SetFunctionGroup,
                       SetValueVelocity := "DB1_DatabaseAgv".MotorDePasso.Inputs.SetValueVelocity,
                       SetValuePosition := "DB1_DatabaseAgv".MotorDePasso.Inputs.SetValuePosition,
                       SetValueForceRamp := "DB1_DatabaseAgv".MotorDePasso.Inputs.SetValueForceRamp,
                       SetValueForce := "DB1_DatabaseAgv".MotorDePasso.Inputs.SetValueForce,
                       SetValueRotRamp := "DB1_DatabaseAgv".MotorDePasso.Inputs.SetValueRotRamp,
                       SetValueRotSpeed := "DB1_DatabaseAgv".MotorDePasso.Inputs.SetValueRotSpeed,
                       FML_REF := #FML_REF,
                       DriveEnabled => "DB1_DatabaseAgv".MotorDePasso.OutPuts.DriveEnabled,
                       Ready => "DB1_DatabaseAgv".MotorDePasso.OutPuts.Ready,
                       Warning => "DB1_DatabaseAgv".MotorDePasso.OutPuts.Warning,
                       Fault => "DB1_DatabaseAgv".MotorDePasso.OutPuts.Fault,
                       SupplyVoltPresent => "DB1_DatabaseAgv".MotorDePasso.OutPuts.SupplyVoltPresent,
                       ControlFCT_HMI => "DB1_DatabaseAgv".MotorDePasso.OutPuts.ControlFCT_HMI,
                       StateOPM => "DB1_DatabaseAgv".MotorDePasso.OutPuts.StateOPM,
                       HaltNotActive => "DB1_DatabaseAgv".MotorDePasso.OutPuts.HaltNotActive,
                       AckStart => "DB1_DatabaseAgv".MotorDePasso.OutPuts.AckStart,
                       MC => "DB1_DatabaseAgv".MotorDePasso.OutPuts.MC,
                       AckTeach => "DB1_DatabaseAgv".MotorDePasso.OutPuts.AckTeach,
                       DriveMoving => "DB1_DatabaseAgv".MotorDePasso.OutPuts.DriveMoving,
                       DragError => "DB1_DatabaseAgv".MotorDePasso.OutPuts.DragError,
                       StandStillControl => "DB1_DatabaseAgv".MotorDePasso.OutPuts.StandStillControl,
                       HomingValid => "DB1_DatabaseAgv".MotorDePasso.OutPuts.HomingValid,
                       ActualRecordNo => "DB1_DatabaseAgv".MotorDePasso.OutPuts.ActualRecordNo,
                       RC1 => "DB1_DatabaseAgv".MotorDePasso.OutPuts.RC1,
                       RCC => "DB1_DatabaseAgv".MotorDePasso.OutPuts.RCC,
                       VelocityLimitReached => "DB1_DatabaseAgv".MotorDePasso.OutPuts.VelocityLimitReached,
                       StrokeLimitReached => "DB1_DatabaseAgv".MotorDePasso.OutPuts.StrokeLimitReached,
                       FunctionIsActive => "DB1_DatabaseAgv".MotorDePasso.OutPuts.FunctionIsActive,
                       ActualFunctionNumber => "DB1_DatabaseAgv".MotorDePasso.OutPuts.ActualFunctionNumber,
                       ActualFunctionGroup => "DB1_DatabaseAgv".MotorDePasso.OutPuts.ActualFunctionGroup,
                       ActualPosition => "DB1_DatabaseAgv".MotorDePasso.OutPuts.ActualPosition,
                       ActualVelocity => "DB1_DatabaseAgv".MotorDePasso.OutPuts.ActualVelocity,
                       ActualForce => "DB1_DatabaseAgv".MotorDePasso.OutPuts.ActualForce,
                       ActualRotRamp => "DB1_DatabaseAgv".MotorDePasso.OutPuts.ActualRotRamp,
                       ActualRotSpeed => "DB1_DatabaseAgv".MotorDePasso.OutPuts.ActualRotSpeed);
END_REGION

REGION Network 3: SET dados no motor de direção
   // Este bloco server para realizar a escrita dos dados no motor de direção
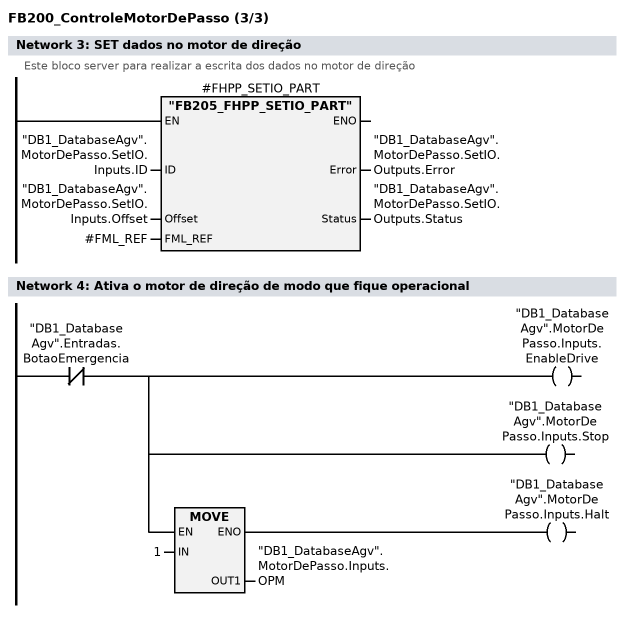
   RUNG wire#powerrail
      #FHPP_SETIO_PART(ID := "DB1_DatabaseAgv".MotorDePasso.SetIO.Inputs.ID, Offset := "DB1_DatabaseAgv".MotorDePasso.SetIO.Inputs.Offset, FML_REF := #FML_REF, Error => "DB1_DatabaseAgv".MotorDePasso.SetIO.Outputs.Error, Status => "DB1_DatabaseAgv".MotorDePasso.SetIO.Outputs.Status)
   END_RUNG
   // the same network as SCL:
   #FHPP_SETIO_PART(ID := "DB1_DatabaseAgv".MotorDePasso.SetIO.Inputs.ID,   // "FB205_FHPP_SETIO_PART"
                    Offset := "DB1_DatabaseAgv".MotorDePasso.SetIO.Inputs.Offset,
                    FML_REF := #FML_REF,
                    Error => "DB1_DatabaseAgv".MotorDePasso.SetIO.Outputs.Error,
                    Status => "DB1_DatabaseAgv".MotorDePasso.SetIO.Outputs.Status);
END_REGION

REGION Network 4: Ativa o motor de direção de modo que fique operacional
   RUNG wire#powerrail
      I_Contact( "DB1_DatabaseAgv".Entradas.BotaoEmergencia )
      wire#w1
      Coil( "DB1_DatabaseAgv".MotorDePasso.Inputs.EnableDrive )
   END_RUNG
   RUNG wire#w1
      Coil( "DB1_DatabaseAgv".MotorDePasso.Inputs.Stop )
   END_RUNG
   RUNG wire#w1
      { S7_GenerateENO := "TRUE" } Move(in := 1, out1 => "DB1_DatabaseAgv".MotorDePasso.Inputs.OPM)
      Coil( "DB1_DatabaseAgv".MotorDePasso.Inputs.Halt )
   END_RUNG
   // the same network as SCL:
   // ENO of a box is taken as its EN; it also drops when the box reports an error
   "DB1_DatabaseAgv".MotorDePasso.Inputs.EnableDrive := NOT "DB1_DatabaseAgv".Entradas.BotaoEmergencia;
   "DB1_DatabaseAgv".MotorDePasso.Inputs.Stop := NOT "DB1_DatabaseAgv".Entradas.BotaoEmergencia;
   IF NOT "DB1_DatabaseAgv".Entradas.BotaoEmergencia THEN
       "DB1_DatabaseAgv".MotorDePasso.Inputs.OPM := 1;
   END_IF;
   "DB1_DatabaseAgv".MotorDePasso.Inputs.Halt := NOT "DB1_DatabaseAgv".Entradas.BotaoEmergencia;
END_REGION
END_FUNCTION_BLOCK

FUNCTION_BLOCK "FB203_FHPP_GETIO_PART"   // FB203, SCL
TITLE = FHPP GETIO_PART
{ S7_Optimized_Access := 'FALSE' }
AUTHOR : FESTO
FAMILY : E-DRIVE
VERSION : 5.1
// Get data from FHPP device using system function GETIO_PART.
   VAR_INPUT
      IAddress_FHPP : Word;
      Offset : Int;   // offset from start address where FHPP data start
      DeviceType : String[16] := 'CMMO_ST';   // CMMO_ST, EMCA_EC, CMMP_AS, CMMS_AS, CMMS_ST, CMMD_AS, SFC_DC, MTR_DCI
   END_VAR
   VAR_OUTPUT
      Error : Bool;   // error while reading
      Status : "DT_FML_STATUS";
   END_VAR
   VAR_IN_OUT
      FML_REF : "DT_FML_REF";
   END_VAR
   VAR
      GET_PART : GETIO_PART;
   END_VAR
   VAR_TEMP
      i : Int;
      iByteCount : DInt;
      tmpFHPPplusSize : DInt;
      tmpFHPPplusElementSize : Array[1..9] of DInt;
      FHPPplus24 : Array[1..24] of Byte;
      tmp : Array[1..9] of DInt;
      WORD_BYTE : Word;
      WBYTE AT WORD_BYTE : Array[1..2] of Byte;
      DWORD_BYTE : DInt;
      DBYTE AT DWORD_BYTE : Array[1..4] of Byte;
      tmpStatus : "DT_FML_STATUS";
      tmp_FML_REF : "DT_FML_REF";
   END_VAR
BEGIN


   // function block (FB) is busy
   #tmpStatus.Err := FALSE;
   #tmpStatus.Cat := 0;
   #tmpStatus.ID :=0; // FB busy 

   // check device type
   IF #DeviceType S_COMP 'CMMO_ST' THEN
       #FML_REF.DeviceTypeNo := 10;
       #FML_REF.DeviceType := #DeviceType;
   ELSE
       #tmpStatus.Err := TRUE;
       #tmpStatus.Cat := 1; // functionblock
       #tmpStatus.ID := DWORD_TO_DINT(16#8000_001E); // device type not valid
   END_IF;

   // ### FHPP Standard ###########################################
   // 

   #GET_PART(ID := #IAddress_FHPP,
             OFFSET := #Offset,
             LEN := 8,
             ERROR => #tmpStatus.Err,
             INPUTS := #FML_REF.InData.FHPP);

   // Error while reading?
   IF #tmpStatus.Err THEN
       #tmpStatus.Cat := 4; // SIEMENS
       #tmpStatus.ID := DWORD_TO_DINT(#GET_PART.STATUS);
   END_IF;



   // ### EXIT ROUTINE ############################################################
   IF NOT #tmpStatus.Err THEN
       ENO := TRUE;      // Set ENO-Bit to true
       #Status := #tmpStatus;
       #Error := #tmpStatus.Err;
   ELSE
       ENO := FALSE;     // Set ENO-Bit to false
       #Status := #tmpStatus;
       #Error := #tmpStatus.Err;
   END_IF;
END_FUNCTION_BLOCK

FUNCTION_BLOCK "FB204_FHPP_CTRL"   // FB204, SCL
TITLE = FHPP_CTRL
{ S7_Optimized_Access := 'FALSE' }
AUTHOR : FESTO
FAMILY : E-DRIVE
VERSION : 5.1
// control FHPP drive
   VAR_INPUT
      EnableDrive : Bool;   // Enable the Drive
      Stop : Bool;   // Stop active == 0 / Stop not active == 1
      Halt : Bool;   // Halt active == 0 / Halt not active == 1
      Brake : Bool;   // Release Brake
      ResetFault : Bool;   // Quit active Fault
      HMIAccessLocked : Bool;   // SPS Control == 1 / HMI Control == 0
      OPM : Int;   // Operation Mode CPOS
      StartTask : Bool;   // Starts Positioning Task
      StartHoming : Bool;   // Starts Homing Task
      JogPos : Bool;   // Jogging positive direction
      JogNeg : Bool;   // Jogging negaitive direction
      TeachActValue : Bool;   // Teach actual position to selected record number
      ClearRemPos : Bool;   // Clear remaining Position if Halt is/was active CDIR
      Relative : Bool;   // Absolute == 0 / Relative == 1
      DeactivateStrokeLimit : Bool;   // deactivate stroke limit (directmode/force-control)
      ExecuteFunction : Bool;   // execute cam disc function(TRUE = execute)
      RecordNo : Int;   // pre selection of the record number (Recordmode)
      SetFunctionNumber : Int;   // set cam disc function number
      SetFunctionGroup : Int;   // set cam disc function group
      SetValueVelocity : DInt;   // Setvalue Velocity (Directmode/Positionmode)
      SetValuePosition : DInt;   // pre selection Position (Directmode/Positioncontrol)
      SetValueForceRamp : DInt;   // actual value for force-ramp (directmode/force-control)
      SetValueForce : DInt;   // Setvalue Force (Directmode/Forcecontrol)
      SetValueRotRamp : DInt;   // Setvalue for Rotation-Speed-Ramp (Directmode/Rotation-Speed-Control)
      SetValueRotSpeed : DInt;   // Setvalue for Rotation-Speed (Directmode/Rotation-Speed-Control)
   END_VAR
   VAR_OUTPUT
      DriveEnabled : Bool;   // 0 == Disabled, 1 == Enabled
      Ready : Bool;   // Drive is Ready
      Warning : Bool;   // indicates Information to user (no Stop of axis)
      Fault : Bool;   // indicates Information to user (Stop of axis)
      SupplyVoltPresent : Bool;   // 0 == not present, 1 == present
      ControlFCT_HMI : Bool;   // 0 == Access MMI, 1 == SPS
      StateOPM : Int;   // State of Operation Mode (INT) SPOS
      HaltNotActive : Bool;   // 1 == Halt is not active
      AckStart : Bool;   // Acknowledge Start
      MC : Bool;   // Motioncomplete
      AckTeach : Bool;   // Acknowledge Teach
      DriveMoving : Bool;   // 1 == Drive is moving
      DragError : Bool;   // 1 == Drag Error active
      StandStillControl : Bool;   // 1 == Axis is outside tolerance window after MC
      HomingValid : Bool;   // Drive is referenced
      ActualRecordNo : Int;   // Actual Recordnumber (Recordmode)
      RC1 : Bool;   // Record Chain Condition 1 reached
      RCC : Bool;   // Record Chain Condition Complete
      VelocityLimitReached : Bool;
      StrokeLimitReached : Bool;
      FunctionIsActive : Bool;   // status of cam disc function
      ActualFunctionNumber : Int;   // actual cam disc function number
      ActualFunctionGroup : Int;   // actual cam disc function group
      ActualPosition : DInt;   // Actual Position (Directmode/Positioncontrol)
      ActualVelocity : Int;   // Actual Velocity (Directmode)
      ActualForce : Int;   // Actual Force (Directmode/Forcecontrol)
      ActualRotRamp : Int;   // Actvalue FOR Rotation-Speed-Ramp (Directmode/Rotation-Speed-Control
      ActualRotSpeed : DInt;   // Actvalue FOR Rotation-Speed (Directmode/Rotation-Speed-Control
   END_VAR
   VAR_IN_OUT
      FML_REF : "DT_FML_REF";
   END_VAR
   VAR
      Converted_BYTE5_8 : DInt;
      BByte AT Converted_BYTE5_8 : Array[1..4] of Byte;
      _Byte : Byte;
      BBit AT _Byte : Array[0..7] of Bool;
      _Word : Word;
      WBit AT _Word : Array[0..15] of Bool;
      OperationModeB1 : Bool;
      OperationModeB2 : Bool;
      ControlModeB1 : Bool;
      ControlModeB2 : Bool;
      ContinuousMode : Bool;
      StateOperationModeB1 : Bool;
      StateOperationModeB2 : Bool;
      StateControlModeB1 : Bool;
      StateControlModeB2 : Bool;
      StateContinuousMode : Bool;
   END_VAR
   VAR_TEMP
      tmpDevice : String[16];
   END_VAR
BEGIN
   (*############################################################
      FESTO AG  Co., Esslingen
      Copyright (c) 2015. All rights reserved.    

      NAME OF FUNCTION BLOCK:         FHPP_CTRL
      VERSION NUMBER:                 V5.1
      COMPOSER:                       bejk


      -----------------------------------------------------
      Date        Name                Activity                                                                              
      15.04.2015  Benjamin Kilgus     converted from Step7 V5.5 (V3.0)
      25.08.2015  Benjamin Kilgus     ActualVelocity, cast changed to BYTE_TO_SINT 
                                      case 5 for SetValue's adjusted to FW specific differents (V3.1)
      16.11.2015  Benjamin Kilgus     Änderungen für kompatibilität S7300/S7400 (V3.2)   
      13.04.2016  Benjamin Klein      Änderungen für FUNC Bit hinzugefügt
      01.08.2016  Benjamin Klein      SetValueForce wird auf 120% begrenzt, da die Rückmeldung nur 1 Byte Wertebereich hat.
      12.08.2016  Benjamin Klein      Datentyp ActualVelocity,ActualForce und ActualRotRamp auf INT geändert. 
      29.08.2016  Benjamin Klein      version changed (V4.1)
      21.09.2016  Benjamin Klein      bugfix Actual Force, limit in SetForce deactivated, SetFunctionNumber bugfix, FML_REF.InData.FHPP[4] in StateOPM changed for S7-300 (V4.2)
      07.07.2017  Benjamin Klein      version chagend (V5.1) - no functional changes
   ############################################################*)

   (*-----------------------------------------------------------
       Initial Block Routine
   ------------------------------------------------------------*)
   #tmpDevice := #FML_REF.DeviceType;

   (* Byte_3 *)
   #StrokeLimitReached := FALSE;
   #VelocityLimitReached := FALSE;
   #StateContinuousMode := FALSE;
   #StateControlModeB2 := FALSE;
   #StateControlModeB1 := FALSE;
   #ActualRecordNo := 0;

   (* Byte_4 *)
   #RC1 := FALSE;
   #RCC := FALSE;
   #VelocityLimitReached := FALSE;
   #StrokeLimitReached := FALSE;

   #ActualVelocity := 0;
   #ActualForce := 0;
   #ActualRotRamp := 0;

   (* Byte5-8 *)
   #ActualPosition := 0;
   #ActualRotSpeed := 0;

   (*-----------------------------------------------------------
       Asignment of the Input Data (Stateword)
   ------------------------------------------------------------*)

   #BByte[1] := #FML_REF.InData.FHPP[5];
   #BByte[2] := #FML_REF.InData.FHPP[6];
   #BByte[3] := #FML_REF.InData.FHPP[7];
   #BByte[4] := #FML_REF.InData.FHPP[8];

   (* Byte1 SCON *)
   #_Byte := #FML_REF.InData.FHPP[1];
   #StateOperationModeB2 := #BBit[7];
   #StateOperationModeB1 := #BBit[6];
   #ControlFCT_HMI := #BBit[5];
   #SupplyVoltPresent := #BBit[4];
   #Fault := #BBit[3];
   #Warning := #BBit[2];
   #Ready := #BBit[1];
   #DriveEnabled := #BBit[0];

   (* Byte2 SPOS *)
   #_Byte := #FML_REF.InData.FHPP[2];
   #HomingValid := #BBit[7];
   #StandStillControl := #BBit[6];
   #DragError := #BBit[5];
   #DriveMoving := #BBit[4];
   #AckTeach := #BBit[3];
   #MC := #BBit[2];
   #AckStart := #BBit[1];
   #HaltNotActive := #BBit[0];

   (* Byte_3 *)
   IF #StateOperationModeB1 THEN        // ===== directmode active =====
   (* SDIR *)
       #_Byte := #FML_REF.InData.FHPP[3];
       IF #BBit[7] AND #tmpDevice S_COMP 'CMMP_AS' THEN

           IF #BBit[3] AND #BBit[4] THEN
               #ActualFunctionNumber := 3;
           ELSIF NOT #BBit[3] AND #BBit[4] THEN
               #ActualFunctionNumber := 2;
           ELSIF #BBit[3] AND NOT #BBit[4] THEN
               #ActualFunctionNumber := 1;
           ELSE
               #ActualFunctionNumber := 0;
           END_IF;

           IF #BBit[5] AND #BBit[6] THEN
               #ActualFunctionGroup := 3;
           ELSIF NOT #BBit[5] AND #BBit[6] THEN
               #ActualFunctionGroup := 2;
           ELSIF #BBit[5] AND NOT #BBit[6] THEN
               #ActualFunctionGroup := 1;
           ELSE
               #ActualFunctionGroup := 0;
           END_IF;

           #FunctionIsActive := TRUE;
           #StateControlModeB2 := #BBit[2];
           #StateControlModeB1 := #BBit[1];
           ;
       ELSE
           #StrokeLimitReached := #BBit[5];
           #VelocityLimitReached := #BBit[4];
           #StateContinuousMode := #BBit[3];
           #StateControlModeB2 := #BBit[2];
           #StateControlModeB1 := #BBit[1];

           #FunctionIsActive := FALSE;
           #ActualFunctionNumber := 0;
           #ActualFunctionGroup := 0;
       END_IF;
   ELSE                                // ===== recordmode active =====
   (* RecordNo *)
       #ActualRecordNo := BYTE_TO_INT(#FML_REF.InData.FHPP[3]);

       #FunctionIsActive := FALSE;
       #ActualFunctionNumber := 0;
       #ActualFunctionGroup := 0;
       ;
   END_IF;

   (* Coding of the Operation Mode State *)
   #_Word := 0;
   #WBit[8] := #StateOperationModeB1;
   #WBit[9] := #StateOperationModeB2;
   #WBit[10] := #StateControlModeB1;
   #WBit[11] := #StateControlModeB2;
   #WBit[12] := #StateContinuousMode;
   #StateOPM := WORD_TO_INT(#_Word);

   (* Byte_4/ Byte5-8*)
   CASE #StateOPM OF
       0:// (0)  Recordmode
           (* RSB record state *)
           #_Byte := #FML_REF.InData.FHPP[4];
           #RC1 := #BBit[0];
           #RCC := #BBit[1];
           #VelocityLimitReached := #BBit[4];
           #StrokeLimitReached := #BBit[5];
           #ActualPosition := #Converted_BYTE5_8;

       1:
           // (1)  Directmode Position Control
           IF BYTE_TO_INT(#FML_REF.InData.FHPP[4]) >= 128 THEN
               #ActualVelocity := BYTE_TO_INT(#FML_REF.InData.FHPP[4] XOR B#16#FF);     // change Value to Positive Transfer to int
               #ActualVelocity := (#ActualVelocity + 1) * (-1);                    // Change to negative again
           ELSE
               #ActualVelocity := BYTE_TO_INT(#FML_REF.InData.FHPP[4]);
           END_IF;

           #ActualPosition := #Converted_BYTE5_8;

       5:// Directmode Force Control 

           IF BYTE_TO_DINT(#FML_REF.InData.FHPP[4]) >= 128 THEN
               #ActualForce := BYTE_TO_INT(#FML_REF.InData.FHPP[4] XOR B#16#FF);     // change Value to Positive Transfer to int
               #ActualForce := (#ActualForce + 1) * (-1);                             // Change to negative again
           ELSE
               #ActualForce := BYTE_TO_INT(#FML_REF.InData.FHPP[4]);
           END_IF;
           #ActualPosition := #Converted_BYTE5_8;

       9:// Directmode Rotation-Speed-Control
           IF BYTE_TO_INT(#FML_REF.InData.FHPP[4]) >= 128 THEN
               #ActualRotRamp := BYTE_TO_INT(#FML_REF.InData.FHPP[4] XOR B#16#FF);     // change Value to Positive Transfer to int
               #ActualRotRamp := (#ActualRotRamp + 1) * (-1);                           // Change to negative again
           ELSE
               #ActualRotRamp := BYTE_TO_INT(#FML_REF.InData.FHPP[4]);
           END_IF;
           #ActualRotSpeed := #Converted_BYTE5_8;

   END_CASE;

   (*-----------------------------------------------------------
       Asignment of the Output Data (Controlword)
   ------------------------------------------------------------*)
   (* Decoding of the Operationmode *)
   #_Word := INT_TO_WORD(#OPM);
   #OperationModeB1 := #WBit[8];
   #OperationModeB2 := #WBit[9];
   #ControlModeB1 := #WBit[10];
   #ControlModeB2 := #WBit[11];
   #ContinuousMode := #WBit[12];

   (* CCON Byte_1 *)
   #_Byte := 0;
   #BBit[7] := #OperationModeB2;
   #BBit[6] := #OperationModeB1; // selection of Operation Mode
   #BBit[5] := #HMIAccessLocked; // get control sovereignty
   #BBit[4] := false;
   #BBit[3] := #ResetFault;
   #BBit[2] := #Brake;
   #BBit[1] := #Stop;
   #BBit[0] := #EnableDrive;
   #FML_REF.OutData.FHPP[1] := #_Byte;

   (* CPOS Byte_2 *)
   #_Byte := 0;
   #BBit[7] := FALSE;
   #BBit[6] := #ClearRemPos;
   #BBit[5] := #TeachActValue;
   #BBit[4] := #JogNeg;
   #BBit[3] := #JogPos;
   #BBit[2] := #StartHoming;
   #BBit[1] := #StartTask;
   #BBit[0] := #Halt;
   #FML_REF.OutData.FHPP[2] := #_Byte;

   (* Byte_3 *)
   IF #OperationModeB1 THEN     // ===== directmode =====
   (* CDIR *)
       IF #ExecuteFunction AND #tmpDevice S_COMP 'CMMP_AS' THEN
           #_Byte := 0;
           #BBit[7] := TRUE;                                          // CDIR_B7:FUNC
           #BBit[6] := false;                                     // Func Group actually not used
           #BBit[5] := false;                                     // Func Group actually not used
           IF #SetFunctionNumber = 3 THEN
               #BBit[4] := TRUE;
               #BBit[3] := TRUE;
           ELSIF #SetFunctionNumber = 2 THEN
               #BBit[4] := TRUE;
               #BBit[3] := FALSE;
           ELSIF #SetFunctionNumber = 1 THEN
               #BBit[4] := FALSE;
               #BBit[3] := TRUE;
           ELSE
               #BBit[4] := FALSE;
               #BBit[3] := false;
           END_IF;
           #BBit[2] := #ControlModeB2;
           #BBit[1] := #ControlModeB1;
           #BBit[0] := #Relative;
           #FML_REF.OutData.FHPP[3] := #_Byte;
       ELSE
           #_Byte := 0;
           #BBit[7] := FALSE;
           #BBit[6] := FALSE;
           #BBit[5] := #DeactivateStrokeLimit;
           #BBit[4] := FALSE;
           #BBit[3] := FALSE;
           #BBit[2] := #ControlModeB2;
           #BBit[1] := #ControlModeB1;
           #BBit[0] := #Relative;
           #FML_REF.OutData.FHPP[3] := #_Byte;
       END_IF;
   ELSE                        // ===== recordmode =====
   (* RecordNo *)
       #FML_REF.OutData.FHPP[3] := INT_TO_BYTE(#RecordNo);
   END_IF;

   (* Byte4/ Byte5-8 *)
   CASE #OPM OF
       0:// (0)  Recordmode
           #FML_REF.OutData.FHPP[4] := 0;
           #Converted_BYTE5_8 := 0;

       1:
           // (1)  Directmode Position Control
           #FML_REF.OutData.FHPP[4] := DINT_TO_BYTE(MIN(IN1 := #SetValueVelocity, IN2 := 100));                   // byte 4 (permissible range of value is 0 to 100)
           #Converted_BYTE5_8 := #SetValuePosition;

       5:// Directmode Forcecontrol
           (* CMMP-AS *)
           IF (#tmpDevice S_COMP 'CMMP_AS') THEN
               #FML_REF.OutData.FHPP[4] := DINT_TO_BYTE(MIN(IN1 := #SetValueForceRamp, IN2 := 100));          // byte 4 (permissible range of value is 0 to 100);
               (* CMMO-ST AND EMCA-EC *)
           ELSIF (#tmpDevice S_COMP 'CMMO_ST') OR (#tmpDevice S_COMP 'EMCA_EC') THEN
               #FML_REF.OutData.FHPP[4] := DINT_TO_BYTE(MIN(IN1 := #SetValueVelocity, IN2 := 100));
               (*other*)
           ELSE
               #FML_REF.OutData.FHPP[4] := 0;
           END_IF;

           #Converted_BYTE5_8 := #SetValueForce;


       9:// Directmode Rotation-Speed-Control      
           #FML_REF.OutData.FHPP[4] := DINT_TO_BYTE(MIN(IN1 := #SetValueRotRamp, IN2 := 100));                     // byte 4 (permissible range of value is 0 to 100)
           #Converted_BYTE5_8 := #SetValueRotSpeed;

